Yaskawa INFORM job: test_long_tjr7.JBI

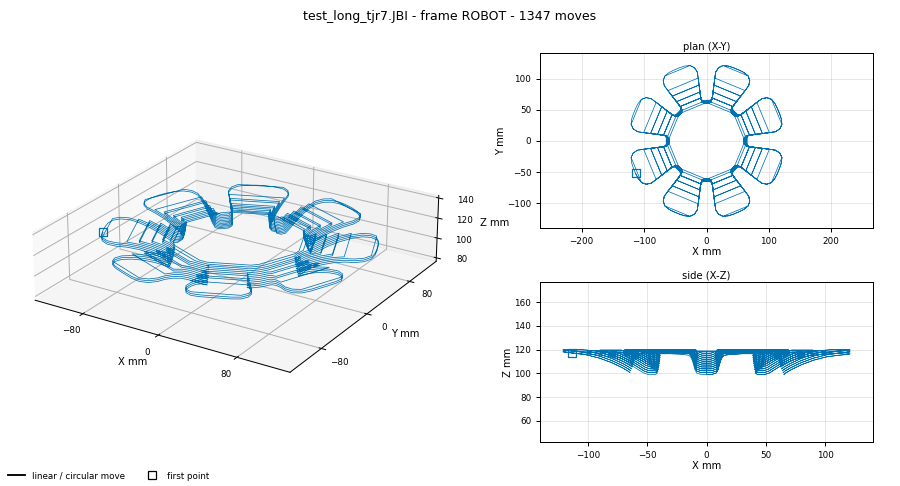
[picture p0: tool path of test_long_tjr7.JBI in frame ROBOT, 1347 of 1348 moves have a stored position in this frame; points joined in program order, loops and branches not executed]
version: 0
/JOB
//NAME test_long
//POS
///NPOS 48,0,0,2,0,0
///TOOL 1
///POSTYPE ROBOT
///RECTAN
///RCONF 1,0,0,0,0,0,0,0,0,0,0,0,0,0,0,0,0,0,0,0,0,0,0,0
C00000=-117.180,-43.520,117.250,-0.0000,-0.0000,1.0000
C00001=-113.630,-52.090,117.250,-0.0000,-0.0000,1.0000
C00002=-109.550,-60.200,116.900,-0.0000,-0.0000,1.0000
C00003=-104.240,-66.670,116.350,-0.0000,-0.0100,1.0000
C00004=-96.760,-69.360,115.810,-0.0000,-0.0200,1.0000
C00005=-88.650,-67.660,115.130,0.0100,-0.0300,1.0000
C00006=-80.860,-61.910,113.810,0.0200,-0.0300,1.0000
C00007=-72.270,-55.220,111.040,0.0200,-0.0300,1.0000
C00008=-64.140,-48.820,107.190,0.0300,-0.0400,1.0000
C00009=-57.630,-43.750,103.240,0.0200,-0.0300,1.0000
C00010=-52.970,-41.300,100.260,-0.0100,0.2100,0.9800
C00011=-49.290,-42.870,99.050,0.2400,0.3300,0.9100
C00012=-47.340,-44.830,99.000,0.3100,0.2900,0.9100
C00013=-46.090,-46.090,99.040,0.3000,0.3000,0.9100
C00014=-44.830,-47.340,99.000,0.2900,0.3100,0.9100
C00015=-42.870,-49.290,99.050,0.3300,0.2400,0.9100
C00016=-41.300,-52.970,100.260,0.2100,-0.0100,0.9800
C00017=-43.750,-57.630,103.240,-0.0300,0.0200,1.0000
C00018=-48.820,-64.140,107.190,-0.0400,0.0300,1.0000
C00019=-55.220,-72.270,111.040,-0.0300,0.0200,1.0000
C00020=-61.910,-80.860,113.810,-0.0300,0.0200,1.0000
C00021=-67.660,-88.650,115.130,-0.0300,0.0100,1.0000
C00022=-69.360,-96.760,115.810,-0.0200,-0.0000,1.0000
C00023=-66.670,-104.240,116.350,-0.0100,-0.0000,1.0000
C00024=-60.200,-109.550,116.900,-0.0000,-0.0000,1.0000
C00025=-52.090,-113.630,117.250,-0.0000,-0.0000,1.0000
C00026=-43.520,-117.180,117.250,-0.0000,-0.0000,1.0000
C00027=-34.900,-120.030,116.900,-0.0000,-0.0000,1.0000
C00028=-26.560,-120.850,116.350,0.0000,-0.0100,1.0000
C00029=-19.380,-117.470,115.810,0.0100,-0.0100,1.0000
C00030=-14.840,-110.530,115.130,0.0300,-0.0100,1.0000
C00031=-13.400,-100.950,113.810,0.0300,-0.0000,1.0000
C00032=-12.060,-90.150,111.040,0.0400,-0.0100,1.0000
C00033=-10.830,-79.870,107.190,0.0400,-0.0100,1.0000
C00034=-9.820,-71.690,103.240,0.0400,-0.0100,1.0000
C00035=-8.250,-66.660,100.260,-0.1600,0.1400,0.9800
C00036=-4.540,-65.170,99.050,-0.0600,0.4000,0.9100
C00037=-1.770,-65.170,99.000,0.0100,0.4200,0.9100
C00038=0.000,-65.190,99.040,-0.0000,0.4200,0.9100
C00039=0.000,-65.190,99.040,-0.0000,0.4200,0.9100
C00040=1.770,-65.170,99.000,-0.0100,0.4200,0.9100
C00041=4.540,-65.170,99.050,0.0600,0.4000,0.9100
C00042=8.250,-66.660,100.260,0.1600,0.1400,0.9800
C00043=9.820,-71.690,103.240,-0.0400,-0.0100,1.0000
C00044=10.830,-79.870,107.190,-0.0400,-0.0100,1.0000
C00045=12.060,-90.150,111.040,-0.0400,-0.0100,1.0000
C00046=13.400,-100.950,113.810,-0.0300,-0.0000,1.0000
C00047=14.840,-110.530,115.130,-0.0300,-0.0100,1.0000
C00048=19.380,-117.470,115.810,-0.0100,-0.0100,1.0000
C00049=26.560,-120.850,116.350,-0.0000,-0.0100,1.0000
C00050=34.900,-120.030,116.900,0.0000,-0.0000,1.0000
C00051=43.520,-117.180,117.250,0.0000,-0.0000,1.0000
C00052=52.090,-113.630,117.250,0.0000,-0.0000,1.0000
C00053=60.200,-109.550,116.900,0.0000,-0.0000,1.0000
C00054=66.670,-104.240,116.350,0.0100,-0.0000,1.0000
C00055=69.360,-96.760,115.810,0.0200,-0.0000,1.0000
C00056=67.660,-88.650,115.130,0.0300,0.0100,1.0000
C00057=61.910,-80.860,113.810,0.0300,0.0200,1.0000
C00058=55.220,-72.270,111.040,0.0300,0.0200,1.0000
C00059=48.820,-64.140,107.190,0.0400,0.0300,1.0000
C00060=43.750,-57.630,103.240,0.0300,0.0200,1.0000
C00061=41.300,-52.970,100.260,-0.2100,-0.0100,0.9800
C00062=42.870,-49.290,99.050,-0.3300,0.2400,0.9100
C00063=44.830,-47.340,99.000,-0.2900,0.3100,0.9100
C00064=46.090,-46.090,99.040,-0.3000,0.3000,0.9100
C00065=47.340,-44.830,99.000,-0.3100,0.2900,0.9100
C00066=49.290,-42.870,99.050,-0.2400,0.3300,0.9100
C00067=52.970,-41.300,100.260,0.0100,0.2100,0.9800
C00068=57.630,-43.750,103.240,-0.0200,-0.0300,1.0000
C00069=64.140,-48.820,107.190,-0.0300,-0.0400,1.0000
C00070=72.270,-55.220,111.040,-0.0200,-0.0300,1.0000
C00071=80.860,-61.910,113.810,-0.0200,-0.0300,1.0000
C00072=88.650,-67.660,115.130,-0.0100,-0.0300,1.0000
C00073=96.760,-69.360,115.810,0.0000,-0.0200,1.0000
C00074=104.240,-66.670,116.350,0.0000,-0.0100,1.0000
C00075=109.550,-60.200,116.900,0.0000,-0.0000,1.0000
C00076=113.630,-52.090,117.250,0.0000,-0.0000,1.0000
C00077=117.180,-43.520,117.250,0.0000,-0.0000,1.0000
C00078=120.030,-34.900,116.900,0.0000,-0.0000,1.0000
C00079=120.850,-26.560,116.350,0.0100,0.0000,1.0000
C00080=117.470,-19.380,115.810,0.0100,0.0100,1.0000
C00081=110.530,-14.840,115.130,0.0100,0.0300,1.0000
C00082=100.950,-13.400,113.810,0.0000,0.0300,1.0000
C00083=90.150,-12.060,111.040,0.0100,0.0400,1.0000
C00084=79.870,-10.830,107.190,0.0100,0.0400,1.0000
C00085=71.690,-9.820,103.240,0.0100,0.0400,1.0000
C00086=66.660,-8.250,100.260,-0.1400,-0.1600,0.9800
C00087=65.170,-4.540,99.050,-0.4000,-0.0600,0.9100
C00088=65.170,-1.770,99.000,-0.4200,0.0100,0.9100
C00089=65.190,0.000,99.040,-0.4200,-0.0000,0.9100
C00090=65.170,1.770,99.000,-0.4200,-0.0100,0.9100
C00091=65.170,4.540,99.050,-0.4000,0.0600,0.9100
C00092=66.660,8.250,100.260,-0.1400,0.1600,0.9800
C00093=71.690,9.820,103.240,0.0100,-0.0400,1.0000
C00094=79.870,10.830,107.190,0.0100,-0.0400,1.0000
C00095=90.150,12.060,111.040,0.0100,-0.0400,1.0000
C00096=100.950,13.400,113.810,0.0000,-0.0300,1.0000
C00097=110.530,14.840,115.130,0.0100,-0.0300,1.0000
C00098=117.470,19.380,115.810,0.0100,-0.0100,1.0000
C00099=120.850,26.560,116.350,0.0100,-0.0000,1.0000
C00100=120.030,34.900,116.900,0.0000,0.0000,1.0000
C00101=117.180,43.520,117.250,0.0000,0.0000,1.0000
C00102=113.630,52.090,117.250,0.0000,0.0000,1.0000
C00103=109.550,60.200,116.900,0.0000,0.0000,1.0000
C00104=104.240,66.670,116.350,0.0000,0.0100,1.0000
C00105=96.760,69.360,115.810,0.0000,0.0200,1.0000
C00106=88.650,67.660,115.130,-0.0100,0.0300,1.0000
C00107=80.860,61.910,113.810,-0.0200,0.0300,1.0000
C00108=72.270,55.220,111.040,-0.0200,0.0300,1.0000
C00109=64.140,48.820,107.190,-0.0300,0.0400,1.0000
C00110=57.630,43.750,103.240,-0.0200,0.0300,1.0000
C00111=52.970,41.300,100.260,0.0100,-0.2100,0.9800
C00112=49.290,42.870,99.050,-0.2400,-0.3300,0.9100
C00113=47.340,44.830,99.000,-0.3100,-0.2900,0.9100
C00114=46.090,46.090,99.040,-0.3000,-0.3000,0.9100
C00115=44.830,47.340,99.000,-0.2900,-0.3100,0.9100
C00116=42.870,49.290,99.050,-0.3300,-0.2400,0.9100
C00117=41.300,52.970,100.260,-0.2100,0.0100,0.9800
C00118=43.750,57.630,103.240,0.0300,-0.0200,1.0000
C00119=48.820,64.140,107.190,0.0400,-0.0300,1.0000
C00120=55.220,72.270,111.040,0.0300,-0.0200,1.0000
C00121=61.910,80.860,113.810,0.0300,-0.0200,1.0000
C00122=67.660,88.650,115.130,0.0300,-0.0100,1.0000
C00123=69.360,96.760,115.810,0.0200,0.0000,1.0000
C00124=66.670,104.240,116.350,0.0100,0.0000,1.0000
C00125=60.200,109.550,116.900,0.0000,0.0000,1.0000
C00126=52.090,113.630,117.250,0.0000,0.0000,1.0000
C00127=43.520,117.180,117.250,0.0000,0.0000,1.0000
C00128=34.900,120.030,116.900,0.0000,0.0000,1.0000
C00129=26.560,120.850,116.350,-0.0000,0.0100,1.0000
C00130=19.380,117.470,115.810,-0.0100,0.0100,1.0000
C00131=14.840,110.530,115.130,-0.0300,0.0100,1.0000
C00132=13.400,100.950,113.810,-0.0300,0.0000,1.0000
C00133=12.060,90.150,111.040,-0.0400,0.0100,1.0000
C00134=10.830,79.870,107.190,-0.0400,0.0100,1.0000
C00135=9.820,71.690,103.240,-0.0400,0.0100,1.0000
C00136=8.250,66.660,100.260,0.1600,-0.1400,0.9800
C00137=4.540,65.170,99.050,0.0600,-0.4000,0.9100
C00138=1.770,65.170,99.000,-0.0100,-0.4200,0.9100
C00139=0.000,65.190,99.040,-0.0000,-0.4200,0.9100
C00140=0.000,64.490,100.590,-0.0000,-0.4000,0.9200
C00141=1.710,64.480,100.550,-0.0100,-0.4000,0.9200
C00142=4.440,64.480,100.600,0.0600,-0.3800,0.9200
C00143=8.120,66.020,101.830,0.1500,-0.1200,0.9800
C00144=9.680,71.190,104.850,-0.0300,0.0000,1.0000
C00145=10.710,79.550,108.860,-0.0400,0.0100,1.0000
C00146=11.970,89.980,112.730,-0.0300,0.0000,1.0000
C00147=13.340,100.880,115.510,-0.0300,0.0000,1.0000
C00148=14.790,110.500,116.830,-0.0200,0.0100,1.0000
C00149=19.340,117.460,117.510,-0.0100,0.0100,1.0000
C00150=26.540,120.860,118.050,-0.0000,0.0000,1.0000
C00151=34.880,120.030,118.600,0.0000,0.0000,1.0000
C00152=43.510,117.180,118.950,0.0000,0.0000,1.0000
C00153=52.090,113.630,118.950,0.0000,0.0000,1.0000
C00154=60.210,109.540,118.600,0.0000,0.0000,1.0000
C00155=66.700,104.220,118.050,0.0000,0.0000,1.0000
C00156=69.380,96.730,117.510,0.0100,0.0000,1.0000
C00157=67.680,88.590,116.830,0.0200,-0.0100,1.0000
C00158=61.900,80.770,115.510,0.0200,-0.0200,1.0000
C00159=55.160,72.090,112.730,0.0300,-0.0200,1.0000
C00160=48.670,63.820,108.860,0.0300,-0.0200,1.0000
C00161=43.490,57.190,104.850,0.0300,-0.0200,1.0000
C00162=40.940,52.430,101.830,-0.1900,0.0200,0.9800
C00163=42.460,48.730,100.600,-0.3100,-0.2300,0.9200
C00164=44.380,46.800,100.550,-0.2700,-0.2900,0.9200
C00165=45.600,45.600,100.590,-0.2800,-0.2800,0.9200
C00166=46.800,44.380,100.550,-0.2900,-0.2700,0.9200
C00167=48.730,42.460,100.600,-0.2300,-0.3100,0.9200
C00168=52.430,40.940,101.830,0.0200,-0.1900,0.9800
C00169=57.190,43.490,104.850,-0.0200,0.0300,1.0000
C00170=63.820,48.670,108.860,-0.0200,0.0300,1.0000
C00171=72.090,55.160,112.730,-0.0200,0.0300,1.0000
C00172=80.770,61.900,115.510,-0.0200,0.0200,1.0000
C00173=88.590,67.680,116.830,-0.0100,0.0200,1.0000
C00174=96.730,69.380,117.510,0.0000,0.0100,1.0000
C00175=104.220,66.700,118.050,0.0000,0.0000,1.0000
C00176=109.540,60.210,118.600,0.0000,0.0000,1.0000
C00177=113.630,52.090,118.950,0.0000,0.0000,1.0000
C00178=117.180,43.510,118.950,0.0000,0.0000,1.0000
C00179=120.030,34.880,118.600,0.0000,0.0000,1.0000
C00180=120.860,26.540,118.050,0.0000,-0.0000,1.0000
C00181=117.460,19.340,117.510,0.0100,-0.0100,1.0000
C00182=110.500,14.790,116.830,0.0100,-0.0200,1.0000
C00183=100.880,13.340,115.510,0.0000,-0.0300,1.0000
C00184=89.980,11.970,112.730,0.0000,-0.0300,1.0000
C00185=79.550,10.710,108.860,0.0100,-0.0400,1.0000
C00186=71.190,9.680,104.850,0.0000,-0.0300,1.0000
C00187=66.020,8.120,101.830,-0.1200,0.1500,0.9800
C00188=64.480,4.440,100.600,-0.3800,0.0600,0.9200
C00189=64.480,1.710,100.550,-0.4000,-0.0100,0.9200
C00190=64.490,0.000,100.590,-0.4000,-0.0000,0.9200
C00191=64.480,-1.710,100.550,-0.4000,0.0100,0.9200
C00192=64.480,-4.440,100.600,-0.3800,-0.0600,0.9200
C00193=66.020,-8.120,101.830,-0.1200,-0.1500,0.9800
C00194=71.190,-9.680,104.850,0.0000,0.0300,1.0000
C00195=79.550,-10.710,108.860,0.0100,0.0400,1.0000
C00196=89.980,-11.970,112.730,0.0000,0.0300,1.0000
C00197=100.880,-13.340,115.510,0.0000,0.0300,1.0000
C00198=110.500,-14.790,116.830,0.0100,0.0200,1.0000
C00199=117.460,-19.340,117.510,0.0100,0.0100,1.0000
C00200=120.860,-26.540,118.050,0.0000,0.0000,1.0000
C00201=120.030,-34.880,118.600,0.0000,-0.0000,1.0000
C00202=117.180,-43.510,118.950,0.0000,-0.0000,1.0000
C00203=113.630,-52.090,118.950,0.0000,-0.0000,1.0000
C00204=109.540,-60.210,118.600,0.0000,-0.0000,1.0000
C00205=104.220,-66.700,118.050,0.0000,-0.0000,1.0000
C00206=96.730,-69.380,117.510,0.0000,-0.0100,1.0000
C00207=88.590,-67.680,116.830,-0.0100,-0.0200,1.0000
C00208=80.770,-61.900,115.510,-0.0200,-0.0200,1.0000
C00209=72.090,-55.160,112.730,-0.0200,-0.0300,1.0000
C00210=63.820,-48.670,108.860,-0.0200,-0.0300,1.0000
C00211=57.190,-43.490,104.850,-0.0200,-0.0300,1.0000
C00212=52.430,-40.940,101.830,0.0200,0.1900,0.9800
C00213=48.730,-42.460,100.600,-0.2300,0.3100,0.9200
C00214=46.800,-44.380,100.550,-0.2900,0.2700,0.9200
C00215=45.600,-45.600,100.590,-0.2800,0.2800,0.9200
C00216=44.380,-46.800,100.550,-0.2700,0.2900,0.9200
C00217=42.460,-48.730,100.600,-0.3100,0.2300,0.9200
C00218=40.940,-52.430,101.830,-0.1900,-0.0200,0.9800
C00219=43.490,-57.190,104.850,0.0300,0.0200,1.0000
C00220=48.670,-63.820,108.860,0.0300,0.0200,1.0000
C00221=55.160,-72.090,112.730,0.0300,0.0200,1.0000
C00222=61.900,-80.770,115.510,0.0200,0.0200,1.0000
C00223=67.680,-88.590,116.830,0.0200,0.0100,1.0000
C00224=69.380,-96.730,117.510,0.0100,-0.0000,1.0000
C00225=66.700,-104.220,118.050,0.0000,-0.0000,1.0000
C00226=60.210,-109.540,118.600,0.0000,-0.0000,1.0000
C00227=52.090,-113.630,118.950,0.0000,-0.0000,1.0000
C00228=43.510,-117.180,118.950,0.0000,-0.0000,1.0000
C00229=34.880,-120.030,118.600,0.0000,-0.0000,1.0000
C00230=26.540,-120.860,118.050,-0.0000,-0.0000,1.0000
C00231=19.340,-117.460,117.510,-0.0100,-0.0100,1.0000
C00232=14.790,-110.500,116.830,-0.0200,-0.0100,1.0000
C00233=13.340,-100.880,115.510,-0.0300,-0.0000,1.0000
C00234=11.970,-89.980,112.730,-0.0300,-0.0000,1.0000
C00235=10.710,-79.550,108.860,-0.0400,-0.0100,1.0000
C00236=9.680,-71.190,104.850,-0.0300,-0.0000,1.0000
C00237=8.120,-66.020,101.830,0.1500,0.1200,0.9800
C00238=4.440,-64.480,100.600,0.0600,0.3800,0.9200
C00239=1.710,-64.480,100.550,-0.0100,0.4000,0.9200
C00240=0.000,-64.490,100.590,-0.0000,0.4000,0.9200
C00241=0.000,-64.490,100.590,-0.0000,0.4000,0.9200
C00242=-1.710,-64.480,100.550,0.0100,0.4000,0.9200
C00243=-4.440,-64.480,100.600,-0.0600,0.3800,0.9200
C00244=-8.120,-66.020,101.830,-0.1500,0.1200,0.9800
C00245=-9.680,-71.190,104.850,0.0300,-0.0000,1.0000
C00246=-10.710,-79.550,108.860,0.0400,-0.0100,1.0000
C00247=-11.970,-89.980,112.730,0.0300,-0.0000,1.0000
C00248=-13.340,-100.880,115.510,0.0300,-0.0000,1.0000
C00249=-14.790,-110.500,116.830,0.0200,-0.0100,1.0000
C00250=-19.340,-117.460,117.510,0.0100,-0.0100,1.0000
C00251=-26.540,-120.860,118.050,0.0000,-0.0000,1.0000
C00252=-34.880,-120.030,118.600,-0.0000,-0.0000,1.0000
C00253=-43.510,-117.180,118.950,-0.0000,-0.0000,1.0000
C00254=-52.090,-113.630,118.950,-0.0000,-0.0000,1.0000
C00255=-60.210,-109.540,118.600,-0.0000,-0.0000,1.0000
C00256=-66.700,-104.220,118.050,-0.0000,-0.0000,1.0000
C00257=-69.380,-96.730,117.510,-0.0100,-0.0000,1.0000
C00258=-67.680,-88.590,116.830,-0.0200,0.0100,1.0000
C00259=-61.900,-80.770,115.510,-0.0200,0.0200,1.0000
C00260=-55.160,-72.090,112.730,-0.0300,0.0200,1.0000
C00261=-48.670,-63.820,108.860,-0.0300,0.0200,1.0000
C00262=-43.490,-57.190,104.850,-0.0300,0.0200,1.0000
C00263=-40.940,-52.430,101.830,0.1900,-0.0200,0.9800
C00264=-42.460,-48.730,100.600,0.3100,0.2300,0.9200
C00265=-44.380,-46.800,100.550,0.2700,0.2900,0.9200
C00266=-45.600,-45.600,100.590,0.2800,0.2800,0.9200
C00267=-46.800,-44.380,100.550,0.2900,0.2700,0.9200
C00268=-48.730,-42.460,100.600,0.2300,0.3100,0.9200
C00269=-52.430,-40.940,101.830,-0.0200,0.1900,0.9800
C00270=-57.190,-43.490,104.850,0.0200,-0.0300,1.0000
C00271=-63.820,-48.670,108.860,0.0200,-0.0300,1.0000
C00272=-72.090,-55.160,112.730,0.0200,-0.0300,1.0000
C00273=-80.770,-61.900,115.510,0.0200,-0.0200,1.0000
C00274=-88.590,-67.680,116.830,0.0100,-0.0200,1.0000
C00275=-96.730,-69.380,117.510,-0.0000,-0.0100,1.0000
C00276=-104.220,-66.700,118.050,-0.0000,-0.0000,1.0000
C00277=-109.540,-60.210,118.600,-0.0000,-0.0000,1.0000
C00278=-113.630,-52.090,118.950,-0.0000,-0.0000,1.0000
C00279=-117.180,-43.510,118.950,-0.0000,-0.0000,1.0000
C00280=-120.030,-34.880,118.600,-0.0000,-0.0000,1.0000
C00281=-120.860,-26.540,118.050,-0.0000,0.0000,1.0000
C00282=-117.460,-19.340,117.510,-0.0100,0.0100,1.0000
C00283=-110.500,-14.790,116.830,-0.0100,0.0200,1.0000
C00284=-100.880,-13.340,115.510,-0.0000,0.0300,1.0000
C00285=-89.980,-11.970,112.730,-0.0000,0.0300,1.0000
C00286=-79.550,-10.710,108.860,-0.0100,0.0400,1.0000
C00287=-71.190,-9.680,104.850,-0.0000,0.0300,1.0000
C00288=-66.020,-8.120,101.830,0.1200,-0.1500,0.9800
C00289=-64.480,-4.440,100.600,0.3800,-0.0600,0.9200
C00290=-64.480,-1.710,100.550,0.4000,0.0100,0.9200
C00291=-64.490,0.000,100.590,0.4000,0.0000,0.9200
C00292=-64.480,1.710,100.550,0.4000,-0.0100,0.9200
C00293=-64.480,4.440,100.600,0.3800,0.0600,0.9200
C00294=-66.020,8.120,101.830,0.1200,0.1500,0.9800
C00295=-71.190,9.680,104.850,-0.0000,-0.0300,1.0000
C00296=-79.550,10.710,108.860,-0.0100,-0.0400,1.0000
C00297=-89.980,11.970,112.730,-0.0000,-0.0300,1.0000
C00298=-100.880,13.340,115.510,-0.0000,-0.0300,1.0000
C00299=-110.500,14.790,116.830,-0.0100,-0.0200,1.0000
C00300=-117.460,19.340,117.510,-0.0100,-0.0100,1.0000
C00301=-120.860,26.540,118.050,-0.0000,-0.0000,1.0000
C00302=-120.030,34.880,118.600,-0.0000,0.0000,1.0000
C00303=-117.180,43.510,118.950,-0.0000,0.0000,1.0000
C00304=-113.630,52.090,118.950,-0.0000,0.0000,1.0000
C00305=-109.540,60.210,118.600,-0.0000,0.0000,1.0000
C00306=-104.220,66.700,118.050,-0.0000,0.0000,1.0000
C00307=-96.730,69.380,117.510,-0.0000,0.0100,1.0000
C00308=-88.590,67.680,116.830,0.0100,0.0200,1.0000
C00309=-80.770,61.900,115.510,0.0200,0.0200,1.0000
C00310=-72.090,55.160,112.730,0.0200,0.0300,1.0000
C00311=-63.820,48.670,108.860,0.0200,0.0300,1.0000
C00312=-57.190,43.490,104.850,0.0200,0.0300,1.0000
C00313=-52.430,40.940,101.830,-0.0200,-0.1900,0.9800
C00314=-48.730,42.460,100.600,0.2300,-0.3100,0.9200
C00315=-46.800,44.380,100.550,0.2900,-0.2700,0.9200
C00316=-45.600,45.600,100.590,0.2800,-0.2800,0.9200
C00317=-44.380,46.800,100.550,0.2700,-0.2900,0.9200
C00318=-42.460,48.730,100.600,0.3100,-0.2300,0.9200
C00319=-40.940,52.430,101.830,0.1900,0.0200,0.9800
C00320=-43.490,57.190,104.850,-0.0300,-0.0200,1.0000
C00321=-48.670,63.820,108.860,-0.0300,-0.0200,1.0000
C00322=-55.160,72.090,112.730,-0.0300,-0.0200,1.0000
C00323=-61.900,80.770,115.510,-0.0200,-0.0200,1.0000
C00324=-67.680,88.590,116.830,-0.0200,-0.0100,1.0000
C00325=-69.380,96.730,117.510,-0.0100,0.0000,1.0000
C00326=-66.700,104.220,118.050,-0.0000,0.0000,1.0000
C00327=-60.210,109.540,118.600,-0.0000,0.0000,1.0000
C00328=-52.090,113.630,118.950,-0.0000,0.0000,1.0000
C00329=-43.510,117.180,118.950,-0.0000,0.0000,1.0000
C00330=-34.880,120.030,118.600,-0.0000,0.0000,1.0000
C00331=-26.540,120.860,118.050,0.0000,0.0000,1.0000
C00332=-19.340,117.460,117.510,0.0100,0.0100,1.0000
C00333=-14.790,110.500,116.830,0.0200,0.0100,1.0000
C00334=-13.340,100.880,115.510,0.0300,0.0000,1.0000
C00335=-11.970,89.980,112.730,0.0300,0.0000,1.0000
C00336=-10.710,79.550,108.860,0.0400,0.0100,1.0000
C00337=-9.680,71.190,104.850,0.0300,0.0000,1.0000
C00338=-8.120,66.020,101.830,-0.1500,-0.1200,0.9800
C00339=-4.440,64.480,100.600,-0.0600,-0.3800,0.9200
C00340=-1.710,64.480,100.550,0.0100,-0.4000,0.9200
C00341=0.000,64.490,100.590,-0.0000,-0.4000,0.9200
C00342=0.000,63.830,102.150,-0.0000,-0.3800,0.9300
C00343=-1.650,63.820,102.110,0.0100,-0.3800,0.9300
C00344=-4.330,63.820,102.170,-0.0600,-0.3600,0.9300
C00345=-8.010,65.430,103.420,-0.1300,-0.1100,0.9800
C00346=-9.560,70.730,106.490,0.0300,0.0000,1.0000
C00347=-10.610,79.260,110.530,0.0300,0.0000,1.0000
C00348=-11.900,89.840,114.420,0.0300,0.0000,1.0000
C00349=-13.300,100.830,117.210,0.0200,0.0000,1.0000
C00350=-14.760,110.480,118.530,0.0100,0.0000,1.0000
C00351=-19.320,117.460,119.210,0.0000,0.0000,1.0000
C00352=-26.530,120.860,119.750,0.0000,0.0000,1.0000
C00353=-66.700,104.220,119.750,-0.0000,0.0000,1.0000
C00354=-69.390,96.720,119.210,-0.0000,0.0000,1.0000
C00355=-67.690,88.560,118.530,-0.0100,-0.0000,1.0000
C00356=-61.890,80.700,117.210,-0.0100,-0.0100,1.0000
C00357=-55.110,71.950,114.420,-0.0200,-0.0200,1.0000
C00358=-48.550,63.550,110.530,-0.0300,-0.0200,1.0000
C00359=-43.250,56.780,106.490,-0.0300,-0.0200,1.0000
C00360=-40.600,51.930,103.420,0.1700,0.0200,0.9800
C00361=-42.070,48.200,102.170,0.2900,-0.2100,0.9300
C00362=-43.960,46.290,102.110,0.2600,-0.2700,0.9300
C00363=-45.130,45.130,102.150,0.2700,-0.2700,0.9300
C00364=-46.290,43.960,102.110,0.2700,-0.2600,0.9300
C00365=-48.200,42.070,102.170,0.2100,-0.2900,0.9300
C00366=-51.930,40.600,103.420,-0.0200,-0.1700,0.9800
C00367=-56.780,43.250,106.490,0.0200,0.0300,1.0000
C00368=-63.550,48.550,110.530,0.0200,0.0300,1.0000
C00369=-71.950,55.110,114.420,0.0200,0.0200,1.0000
C00370=-80.700,61.890,117.210,0.0100,0.0100,1.0000
C00371=-88.560,67.690,118.530,0.0000,0.0100,1.0000
C00372=-96.720,69.390,119.210,-0.0000,0.0000,1.0000
C00373=-104.220,66.700,119.750,-0.0000,0.0000,1.0000
C00374=-120.860,26.530,119.750,-0.0000,-0.0000,1.0000
C00375=-117.460,19.320,119.210,-0.0000,-0.0000,1.0000
C00376=-110.480,14.760,118.530,-0.0000,-0.0100,1.0000
C00377=-100.830,13.300,117.210,-0.0000,-0.0200,1.0000
C00378=-89.840,11.900,114.420,-0.0000,-0.0300,1.0000
C00379=-79.260,10.610,110.530,-0.0000,-0.0300,1.0000
C00380=-70.730,9.560,106.490,-0.0000,-0.0300,1.0000
C00381=-65.430,8.010,103.420,0.1100,0.1300,0.9800
C00382=-63.820,4.330,102.170,0.3600,0.0600,0.9300
C00383=-63.820,1.650,102.110,0.3800,-0.0100,0.9300
C00384=-63.830,0.000,102.150,0.3800,0.0000,0.9300
C00385=-63.820,-1.650,102.110,0.3800,0.0100,0.9300
C00386=-63.820,-4.330,102.170,0.3600,-0.0600,0.9300
C00387=-65.430,-8.010,103.420,0.1100,-0.1300,0.9800
C00388=-70.730,-9.560,106.490,-0.0000,0.0300,1.0000
C00389=-79.260,-10.610,110.530,-0.0000,0.0300,1.0000
C00390=-89.840,-11.900,114.420,-0.0000,0.0300,1.0000
C00391=-100.830,-13.300,117.210,-0.0000,0.0200,1.0000
C00392=-110.480,-14.760,118.530,-0.0000,0.0100,1.0000
C00393=-117.460,-19.320,119.210,-0.0000,0.0000,1.0000
C00394=-120.860,-26.530,119.750,-0.0000,0.0000,1.0000
C00395=-104.220,-66.700,119.750,-0.0000,-0.0000,1.0000
C00396=-96.720,-69.390,119.210,-0.0000,-0.0000,1.0000
C00397=-88.560,-67.690,118.530,0.0000,-0.0100,1.0000
C00398=-80.700,-61.890,117.210,0.0100,-0.0100,1.0000
C00399=-71.950,-55.110,114.420,0.0200,-0.0200,1.0000
C00400=-63.550,-48.550,110.530,0.0200,-0.0300,1.0000
C00401=-56.780,-43.250,106.490,0.0200,-0.0300,1.0000
C00402=-51.930,-40.600,103.420,-0.0200,0.1700,0.9800
C00403=-48.200,-42.070,102.170,0.2100,0.2900,0.9300
C00404=-46.290,-43.960,102.110,0.2700,0.2600,0.9300
C00405=-45.130,-45.130,102.150,0.2700,0.2700,0.9300
C00406=-43.960,-46.290,102.110,0.2600,0.2700,0.9300
C00407=-42.070,-48.200,102.170,0.2900,0.2100,0.9300
C00408=-40.600,-51.930,103.420,0.1700,-0.0200,0.9800
C00409=-43.250,-56.780,106.490,-0.0300,0.0200,1.0000
C00410=-48.550,-63.550,110.530,-0.0300,0.0200,1.0000
C00411=-55.110,-71.950,114.420,-0.0200,0.0200,1.0000
C00412=-61.890,-80.700,117.210,-0.0100,0.0100,1.0000
C00413=-67.690,-88.560,118.530,-0.0100,0.0000,1.0000
C00414=-69.390,-96.720,119.210,-0.0000,-0.0000,1.0000
C00415=-66.700,-104.220,119.750,-0.0000,-0.0000,1.0000
C00416=-26.530,-120.860,119.750,0.0000,-0.0000,1.0000
C00417=-19.320,-117.460,119.210,0.0000,-0.0000,1.0000
C00418=-14.760,-110.480,118.530,0.0100,-0.0000,1.0000
C00419=-13.300,-100.830,117.210,0.0200,-0.0000,1.0000
C00420=-11.900,-89.840,114.420,0.0300,-0.0000,1.0000
C00421=-10.610,-79.260,110.530,0.0300,-0.0000,1.0000
C00422=-9.560,-70.730,106.490,0.0300,-0.0000,1.0000
C00423=-8.010,-65.430,103.420,-0.1300,0.1100,0.9800
C00424=-4.330,-63.820,102.170,-0.0600,0.3600,0.9300
C00425=-1.650,-63.820,102.110,0.0100,0.3800,0.9300
C00426=0.000,-63.830,102.150,-0.0000,0.3800,0.9300
C00427=0.000,-63.830,102.150,-0.0000,0.3800,0.9300
C00428=1.650,-63.820,102.110,-0.0100,0.3800,0.9300
C00429=4.330,-63.820,102.170,0.0600,0.3600,0.9300
C00430=8.010,-65.430,103.420,0.1300,0.1100,0.9800
C00431=9.560,-70.730,106.490,-0.0300,-0.0000,1.0000
C00432=10.610,-79.260,110.530,-0.0300,-0.0000,1.0000
C00433=11.900,-89.840,114.420,-0.0300,-0.0000,1.0000
C00434=13.300,-100.830,117.210,-0.0200,-0.0000,1.0000
C00435=14.760,-110.480,118.530,-0.0100,-0.0000,1.0000
C00436=19.320,-117.460,119.210,-0.0000,-0.0000,1.0000
C00437=26.530,-120.860,119.750,-0.0000,-0.0000,1.0000
C00438=66.700,-104.220,119.750,0.0000,-0.0000,1.0000
C00439=69.390,-96.720,119.210,0.0000,-0.0000,1.0000
C00440=67.690,-88.560,118.530,0.0100,0.0000,1.0000
C00441=61.890,-80.700,117.210,0.0100,0.0100,1.0000
C00442=55.110,-71.950,114.420,0.0200,0.0200,1.0000
C00443=48.550,-63.550,110.530,0.0300,0.0200,1.0000
C00444=43.250,-56.780,106.490,0.0300,0.0200,1.0000
C00445=40.600,-51.930,103.420,-0.1700,-0.0200,0.9800
C00446=42.070,-48.200,102.170,-0.2900,0.2100,0.9300
C00447=43.960,-46.290,102.110,-0.2600,0.2700,0.9300
C00448=45.130,-45.130,102.150,-0.2700,0.2700,0.9300
C00449=46.290,-43.960,102.110,-0.2700,0.2600,0.9300
C00450=48.200,-42.070,102.170,-0.2100,0.2900,0.9300
C00451=51.930,-40.600,103.420,0.0200,0.1700,0.9800
C00452=56.780,-43.250,106.490,-0.0200,-0.0300,1.0000
C00453=63.550,-48.550,110.530,-0.0200,-0.0300,1.0000
C00454=71.950,-55.110,114.420,-0.0200,-0.0200,1.0000
C00455=80.700,-61.890,117.210,-0.0100,-0.0100,1.0000
C00456=88.560,-67.690,118.530,-0.0000,-0.0100,1.0000
C00457=96.720,-69.390,119.210,0.0000,-0.0000,1.0000
C00458=104.220,-66.700,119.750,0.0000,-0.0000,1.0000
C00459=120.860,-26.530,119.750,0.0000,0.0000,1.0000
C00460=117.460,-19.320,119.210,0.0000,0.0000,1.0000
C00461=110.480,-14.760,118.530,0.0000,0.0100,1.0000
C00462=100.830,-13.300,117.210,0.0000,0.0200,1.0000
C00463=89.840,-11.900,114.420,0.0000,0.0300,1.0000
C00464=79.260,-10.610,110.530,0.0000,0.0300,1.0000
C00465=70.730,-9.560,106.490,0.0000,0.0300,1.0000
C00466=65.430,-8.010,103.420,-0.1100,-0.1300,0.9800
C00467=63.820,-4.330,102.170,-0.3600,-0.0600,0.9300
C00468=63.820,-1.650,102.110,-0.3800,0.0100,0.9300
C00469=63.830,0.000,102.150,-0.3800,-0.0000,0.9300
C00470=63.820,1.650,102.110,-0.3800,-0.0100,0.9300
C00471=63.820,4.330,102.170,-0.3600,0.0600,0.9300
C00472=65.430,8.010,103.420,-0.1100,0.1300,0.9800
C00473=70.730,9.560,106.490,0.0000,-0.0300,1.0000
C00474=79.260,10.610,110.530,0.0000,-0.0300,1.0000
C00475=89.840,11.900,114.420,0.0000,-0.0300,1.0000
C00476=100.830,13.300,117.210,0.0000,-0.0200,1.0000
C00477=110.480,14.760,118.530,0.0000,-0.0100,1.0000
C00478=117.460,19.320,119.210,0.0000,-0.0000,1.0000
C00479=120.860,26.530,119.750,0.0000,-0.0000,1.0000
C00480=104.220,66.700,119.750,0.0000,0.0000,1.0000
C00481=96.720,69.390,119.210,0.0000,0.0000,1.0000
C00482=88.560,67.690,118.530,-0.0000,0.0100,1.0000
C00483=80.700,61.890,117.210,-0.0100,0.0100,1.0000
C00484=71.950,55.110,114.420,-0.0200,0.0200,1.0000
C00485=63.550,48.550,110.530,-0.0200,0.0300,1.0000
C00486=56.780,43.250,106.490,-0.0200,0.0300,1.0000
C00487=51.930,40.600,103.420,0.0200,-0.1700,0.9800
C00488=48.200,42.070,102.170,-0.2100,-0.2900,0.9300
C00489=46.290,43.960,102.110,-0.2700,-0.2600,0.9300
C00490=45.130,45.130,102.150,-0.2700,-0.2700,0.9300
C00491=43.960,46.290,102.110,-0.2600,-0.2700,0.9300
C00492=42.070,48.200,102.170,-0.2900,-0.2100,0.9300
C00493=40.600,51.930,103.420,-0.1700,0.0200,0.9800
C00494=43.250,56.780,106.490,0.0300,-0.0200,1.0000
C00495=48.550,63.550,110.530,0.0300,-0.0200,1.0000
C00496=55.110,71.950,114.420,0.0200,-0.0200,1.0000
C00497=61.890,80.700,117.210,0.0100,-0.0100,1.0000
C00498=67.690,88.560,118.530,0.0100,-0.0000,1.0000
C00499=69.390,96.720,119.210,0.0000,0.0000,1.0000
C00500=66.700,104.220,119.750,0.0000,0.0000,1.0000
C00501=26.530,120.860,119.750,-0.0000,0.0000,1.0000
C00502=19.320,117.460,119.210,-0.0000,0.0000,1.0000
C00503=14.760,110.480,118.530,-0.0100,0.0000,1.0000
C00504=13.300,100.830,117.210,-0.0200,0.0000,1.0000
C00505=11.900,89.840,114.420,-0.0300,0.0000,1.0000
C00506=10.610,79.260,110.530,-0.0300,0.0000,1.0000
C00507=9.560,70.730,106.490,-0.0300,0.0000,1.0000
C00508=8.010,65.430,103.420,0.1300,-0.1100,0.9800
C00509=4.330,63.820,102.170,0.0600,-0.3600,0.9300
C00510=1.650,63.820,102.110,-0.0100,-0.3800,0.9300
C00511=0.000,63.830,102.150,-0.0000,-0.3800,0.9300
C00512=0.000,63.210,103.730,-0.0000,-0.3500,0.9400
C00513=1.590,63.200,103.700,-0.0100,-0.3500,0.9400
C00514=4.240,63.210,103.750,0.0500,-0.3300,0.9400
C00515=7.900,64.870,105.020,0.1200,-0.1000,0.9900
C00516=9.450,70.320,108.130,-0.0300,0.0000,1.0000
C00517=10.520,79.020,112.210,-0.0300,0.0000,1.0000
C00518=11.850,89.740,116.120,-0.0200,0.0000,1.0000
C00519=13.270,100.800,118.910,-0.0100,0.0000,1.0000
C00520=61.890,80.660,118.910,0.0100,-0.0000,1.0000
C00521=55.080,71.840,116.120,0.0100,-0.0100,1.0000
C00522=48.440,63.320,112.210,0.0200,-0.0200,1.0000
C00523=43.040,56.410,108.130,0.0200,-0.0200,1.0000
C00524=40.290,51.460,105.020,-0.1600,0.0200,0.9900
C00525=41.700,47.690,103.750,-0.2700,-0.2000,0.9400
C00526=43.560,45.810,103.700,-0.2400,-0.2600,0.9400
C00527=44.690,44.690,103.730,-0.2500,-0.2500,0.9400
C00528=45.810,43.560,103.700,-0.2600,-0.2400,0.9400
C00529=47.700,41.700,103.750,-0.2000,-0.2700,0.9400
C00530=51.460,40.290,105.020,0.0200,-0.1600,0.9900
C00531=56.410,43.040,108.130,-0.0200,0.0200,1.0000
C00532=63.320,48.440,112.210,-0.0200,0.0200,1.0000
C00533=71.840,55.080,116.120,-0.0100,0.0100,1.0000
C00534=80.660,61.890,118.910,-0.0000,0.0100,1.0000
C00535=100.800,13.270,118.910,0.0000,-0.0100,1.0000
C00536=89.740,11.850,116.120,0.0000,-0.0200,1.0000
C00537=79.020,10.520,112.210,0.0000,-0.0300,1.0000
C00538=70.320,9.450,108.130,0.0000,-0.0300,1.0000
C00539=64.870,7.900,105.020,-0.1000,0.1200,0.9900
C00540=63.210,4.240,103.750,-0.3300,0.0500,0.9400
C00541=63.200,1.590,103.700,-0.3500,-0.0100,0.9400
C00542=63.210,0.000,103.730,-0.3500,-0.0000,0.9400
C00543=63.200,-1.590,103.700,-0.3500,0.0100,0.9400
C00544=63.210,-4.240,103.750,-0.3300,-0.0500,0.9400
C00545=64.870,-7.900,105.020,-0.1000,-0.1200,0.9900
C00546=70.320,-9.450,108.130,0.0000,0.0300,1.0000
C00547=79.020,-10.520,112.210,0.0000,0.0300,1.0000
C00548=89.740,-11.850,116.120,0.0000,0.0200,1.0000
C00549=100.800,-13.270,118.910,0.0000,0.0100,1.0000
C00550=80.660,-61.890,118.910,-0.0000,-0.0100,1.0000
C00551=71.840,-55.080,116.120,-0.0100,-0.0100,1.0000
C00552=63.320,-48.440,112.210,-0.0200,-0.0200,1.0000
C00553=56.410,-43.040,108.130,-0.0200,-0.0200,1.0000
C00554=51.460,-40.290,105.020,0.0200,0.1600,0.9900
C00555=47.690,-41.700,103.750,-0.2000,0.2700,0.9400
C00556=45.810,-43.560,103.700,-0.2600,0.2400,0.9400
C00557=44.690,-44.690,103.730,-0.2500,0.2500,0.9400
C00558=43.560,-45.810,103.700,-0.2400,0.2600,0.9400
C00559=41.700,-47.700,103.750,-0.2700,0.2000,0.9400
C00560=40.290,-51.460,105.020,-0.1600,-0.0200,0.9900
C00561=43.040,-56.410,108.130,0.0200,0.0200,1.0000
C00562=48.440,-63.320,112.210,0.0200,0.0200,1.0000
C00563=55.080,-71.840,116.120,0.0100,0.0100,1.0000
C00564=61.890,-80.660,118.910,0.0100,0.0000,1.0000
C00565=13.270,-100.800,118.910,-0.0100,-0.0000,1.0000
C00566=11.850,-89.740,116.120,-0.0200,-0.0000,1.0000
C00567=10.520,-79.020,112.210,-0.0300,-0.0000,1.0000
C00568=9.450,-70.320,108.130,-0.0300,-0.0000,1.0000
C00569=7.900,-64.870,105.020,0.1200,0.1000,0.9900
C00570=4.240,-63.210,103.750,0.0500,0.3300,0.9400
C00571=1.590,-63.200,103.700,-0.0100,0.3500,0.9400
C00572=0.000,-63.210,103.730,-0.0000,0.3500,0.9400
C00573=0.000,-63.210,103.730,-0.0000,0.3500,0.9400
C00574=-1.590,-63.200,103.700,0.0100,0.3500,0.9400
C00575=-4.240,-63.210,103.750,-0.0500,0.3300,0.9400
C00576=-7.900,-64.870,105.020,-0.1200,0.1000,0.9900
C00577=-9.450,-70.320,108.130,0.0300,-0.0000,1.0000
C00578=-10.520,-79.020,112.210,0.0300,-0.0000,1.0000
C00579=-11.850,-89.740,116.120,0.0200,-0.0000,1.0000
C00580=-13.270,-100.800,118.910,0.0100,-0.0000,1.0000
C00581=-61.890,-80.660,118.910,-0.0100,0.0000,1.0000
C00582=-55.080,-71.840,116.120,-0.0100,0.0100,1.0000
C00583=-48.440,-63.320,112.210,-0.0200,0.0200,1.0000
C00584=-43.040,-56.410,108.130,-0.0200,0.0200,1.0000
C00585=-40.290,-51.460,105.020,0.1600,-0.0200,0.9900
C00586=-41.700,-47.690,103.750,0.2700,0.2000,0.9400
C00587=-43.560,-45.810,103.700,0.2400,0.2600,0.9400
C00588=-44.690,-44.690,103.730,0.2500,0.2500,0.9400
C00589=-45.810,-43.560,103.700,0.2600,0.2400,0.9400
C00590=-47.700,-41.700,103.750,0.2000,0.2700,0.9400
C00591=-51.460,-40.290,105.020,-0.0200,0.1600,0.9900
C00592=-56.410,-43.040,108.130,0.0200,-0.0200,1.0000
C00593=-63.320,-48.440,112.210,0.0200,-0.0200,1.0000
C00594=-71.840,-55.080,116.120,0.0100,-0.0100,1.0000
C00595=-80.660,-61.890,118.910,0.0000,-0.0100,1.0000
C00596=-100.800,-13.270,118.910,-0.0000,0.0100,1.0000
C00597=-89.740,-11.850,116.120,-0.0000,0.0200,1.0000
C00598=-79.020,-10.520,112.210,-0.0000,0.0300,1.0000
C00599=-70.320,-9.450,108.130,-0.0000,0.0300,1.0000
C00600=-64.870,-7.900,105.020,0.1000,-0.1200,0.9900
C00601=-63.210,-4.240,103.750,0.3300,-0.0500,0.9400
C00602=-63.200,-1.590,103.700,0.3500,0.0100,0.9400
C00603=-63.210,0.000,103.730,0.3500,0.0000,0.9400
C00604=-63.200,1.590,103.700,0.3500,-0.0100,0.9400
C00605=-63.210,4.240,103.750,0.3300,0.0500,0.9400
C00606=-64.870,7.900,105.020,0.1000,0.1200,0.9900
C00607=-70.320,9.450,108.130,-0.0000,-0.0300,1.0000
C00608=-79.020,10.520,112.210,-0.0000,-0.0300,1.0000
C00609=-89.740,11.850,116.120,-0.0000,-0.0200,1.0000
C00610=-100.800,13.270,118.910,-0.0000,-0.0100,1.0000
C00611=-80.660,61.890,118.910,0.0000,0.0100,1.0000
C00612=-71.840,55.080,116.120,0.0100,0.0100,1.0000
C00613=-63.320,48.440,112.210,0.0200,0.0200,1.0000
C00614=-56.410,43.040,108.130,0.0200,0.0200,1.0000
C00615=-51.460,40.290,105.020,-0.0200,-0.1600,0.9900
C00616=-47.690,41.700,103.750,0.2000,-0.2700,0.9400
C00617=-45.810,43.560,103.700,0.2600,-0.2400,0.9400
C00618=-44.690,44.690,103.730,0.2500,-0.2500,0.9400
C00619=-43.560,45.810,103.700,0.2400,-0.2600,0.9400
C00620=-41.700,47.700,103.750,0.2700,-0.2000,0.9400
C00621=-40.290,51.460,105.020,0.1600,0.0200,0.9900
C00622=-43.040,56.410,108.130,-0.0200,-0.0200,1.0000
C00623=-48.440,63.320,112.210,-0.0200,-0.0200,1.0000
C00624=-55.080,71.840,116.120,-0.0100,-0.0100,1.0000
C00625=-61.890,80.660,118.910,-0.0100,-0.0000,1.0000
C00626=-13.270,100.800,118.910,0.0100,0.0000,1.0000
C00627=-11.850,89.740,116.120,0.0200,0.0000,1.0000
C00628=-10.520,79.020,112.210,0.0300,0.0000,1.0000
C00629=-9.450,70.320,108.130,0.0300,0.0000,1.0000
C00630=-7.900,64.870,105.020,-0.1200,-0.1000,0.9900
C00631=-4.240,63.210,103.750,-0.0500,-0.3300,0.9400
C00632=-1.590,63.200,103.700,0.0100,-0.3500,0.9400
C00633=0.000,63.210,103.730,-0.0000,-0.3500,0.9400
C00634=0.000,62.630,105.330,-0.0000,-0.3300,0.9500
C00635=-1.540,62.620,105.300,0.0100,-0.3300,0.9500
C00636=-4.150,62.640,105.350,-0.0500,-0.3100,0.9500
C00637=-7.800,64.360,106.640,-0.1100,-0.0900,0.9900
C00638=-9.350,69.950,109.790,0.0300,0.0000,1.0000
C00639=-10.450,78.820,113.900,0.0200,0.0000,1.0000
C00640=-11.820,89.670,117.820,0.0100,0.0000,1.0000
C00641=-55.050,71.770,117.820,-0.0100,-0.0100,1.0000
C00642=-48.350,63.130,113.900,-0.0200,-0.0100,1.0000
C00643=-42.850,56.080,109.790,-0.0200,-0.0200,1.0000
C00644=-40.000,51.030,106.640,0.1400,0.0100,0.9900
C00645=-41.360,47.230,105.350,0.2500,-0.1800,0.9500
C00646=-43.190,45.370,105.300,0.2200,-0.2400,0.9500
C00647=-44.290,44.290,105.330,0.2300,-0.2300,0.9500
C00648=-45.370,43.190,105.300,0.2400,-0.2200,0.9500
C00649=-47.230,41.360,105.350,0.1800,-0.2500,0.9500
C00650=-51.030,40.000,106.640,-0.0100,-0.1400,0.9900
C00651=-56.080,42.850,109.790,0.0200,0.0200,1.0000
C00652=-63.130,48.350,113.900,0.0100,0.0200,1.0000
C00653=-71.770,55.050,117.820,0.0100,0.0100,1.0000
C00654=-89.670,11.820,117.820,-0.0000,-0.0100,1.0000
C00655=-78.820,10.450,113.900,-0.0000,-0.0200,1.0000
C00656=-69.950,9.350,109.790,-0.0000,-0.0300,1.0000
C00657=-64.360,7.800,106.640,0.0900,0.1100,0.9900
C00658=-62.640,4.150,105.350,0.3100,0.0500,0.9500
C00659=-62.620,1.540,105.300,0.3300,-0.0100,0.9500
C00660=-62.630,0.000,105.330,0.3300,0.0000,0.9500
C00661=-62.620,-1.540,105.300,0.3300,0.0100,0.9500
C00662=-62.640,-4.150,105.350,0.3100,-0.0500,0.9500
C00663=-64.360,-7.800,106.640,0.0900,-0.1100,0.9900
C00664=-69.950,-9.350,109.790,-0.0000,0.0300,1.0000
C00665=-78.820,-10.450,113.900,-0.0000,0.0200,1.0000
C00666=-89.670,-11.820,117.820,-0.0000,0.0100,1.0000
C00667=-71.770,-55.050,117.820,0.0100,-0.0100,1.0000
C00668=-63.130,-48.350,113.900,0.0100,-0.0200,1.0000
C00669=-56.080,-42.850,109.790,0.0200,-0.0200,1.0000
C00670=-51.030,-40.000,106.640,-0.0100,0.1400,0.9900
C00671=-47.230,-41.360,105.350,0.1800,0.2500,0.9500
C00672=-45.370,-43.190,105.300,0.2400,0.2200,0.9500
C00673=-44.290,-44.290,105.330,0.2300,0.2300,0.9500
C00674=-43.190,-45.370,105.300,0.2200,0.2400,0.9500
C00675=-41.360,-47.230,105.350,0.2500,0.1800,0.9500
C00676=-40.000,-51.030,106.640,0.1400,-0.0100,0.9900
C00677=-42.850,-56.080,109.790,-0.0200,0.0200,1.0000
C00678=-48.350,-63.130,113.900,-0.0200,0.0100,1.0000
C00679=-55.050,-71.770,117.820,-0.0100,0.0100,1.0000
C00680=-11.820,-89.670,117.820,0.0100,-0.0000,1.0000
C00681=-10.450,-78.820,113.900,0.0200,-0.0000,1.0000
C00682=-9.350,-69.950,109.790,0.0300,-0.0000,1.0000
C00683=-7.800,-64.360,106.640,-0.1100,0.0900,0.9900
C00684=-4.150,-62.640,105.350,-0.0500,0.3100,0.9500
C00685=-1.540,-62.620,105.300,0.0100,0.3300,0.9500
C00686=0.000,-62.630,105.330,-0.0000,0.3300,0.9500
C00687=0.000,-62.630,105.330,-0.0000,0.3300,0.9500
C00688=1.540,-62.620,105.300,-0.0100,0.3300,0.9500
C00689=4.150,-62.640,105.350,0.0500,0.3100,0.9500
C00690=7.800,-64.360,106.640,0.1100,0.0900,0.9900
C00691=9.350,-69.950,109.790,-0.0300,-0.0000,1.0000
C00692=10.450,-78.820,113.900,-0.0200,-0.0000,1.0000
C00693=11.820,-89.670,117.820,-0.0100,-0.0000,1.0000
C00694=55.050,-71.770,117.820,0.0100,0.0100,1.0000
C00695=48.350,-63.130,113.900,0.0200,0.0100,1.0000
C00696=42.850,-56.080,109.790,0.0200,0.0200,1.0000
C00697=40.000,-51.030,106.640,-0.1400,-0.0100,0.9900
C00698=41.360,-47.230,105.350,-0.2500,0.1800,0.9500
C00699=43.190,-45.370,105.300,-0.2200,0.2400,0.9500
C00700=44.290,-44.290,105.330,-0.2300,0.2300,0.9500
C00701=45.370,-43.190,105.300,-0.2400,0.2200,0.9500
C00702=47.230,-41.360,105.350,-0.1800,0.2500,0.9500
C00703=51.030,-40.000,106.640,0.0100,0.1400,0.9900
C00704=56.080,-42.850,109.790,-0.0200,-0.0200,1.0000
C00705=63.130,-48.350,113.900,-0.0100,-0.0200,1.0000
C00706=71.770,-55.050,117.820,-0.0100,-0.0100,1.0000
C00707=89.670,-11.820,117.820,0.0000,0.0100,1.0000
C00708=78.820,-10.450,113.900,0.0000,0.0200,1.0000
C00709=69.950,-9.350,109.790,0.0000,0.0300,1.0000
C00710=64.360,-7.800,106.640,-0.0900,-0.1100,0.9900
C00711=62.640,-4.150,105.350,-0.3100,-0.0500,0.9500
C00712=62.620,-1.540,105.300,-0.3300,0.0100,0.9500
C00713=62.630,0.000,105.330,-0.3300,-0.0000,0.9500
C00714=62.620,1.540,105.300,-0.3300,-0.0100,0.9500
C00715=62.640,4.150,105.350,-0.3100,0.0500,0.9500
C00716=64.360,7.800,106.640,-0.0900,0.1100,0.9900
C00717=69.950,9.350,109.790,0.0000,-0.0300,1.0000
C00718=78.820,10.450,113.900,0.0000,-0.0200,1.0000
C00719=89.670,11.820,117.820,0.0000,-0.0100,1.0000
C00720=71.770,55.050,117.820,-0.0100,0.0100,1.0000
C00721=63.130,48.350,113.900,-0.0100,0.0200,1.0000
C00722=56.080,42.850,109.790,-0.0200,0.0200,1.0000
C00723=51.030,40.000,106.640,0.0100,-0.1400,0.9900
C00724=47.230,41.360,105.350,-0.1800,-0.2500,0.9500
C00725=45.370,43.190,105.300,-0.2400,-0.2200,0.9500
C00726=44.290,44.290,105.330,-0.2300,-0.2300,0.9500
C00727=43.190,45.370,105.300,-0.2200,-0.2400,0.9500
C00728=41.360,47.230,105.350,-0.2500,-0.1800,0.9500
C00729=40.000,51.030,106.640,-0.1400,0.0100,0.9900
C00730=42.850,56.080,109.790,0.0200,-0.0200,1.0000
C00731=48.350,63.130,113.900,0.0200,-0.0100,1.0000
C00732=55.050,71.770,117.820,0.0100,-0.0100,1.0000
C00733=11.820,89.670,117.820,-0.0100,0.0000,1.0000
C00734=10.450,78.820,113.900,-0.0200,0.0000,1.0000
C00735=9.350,69.950,109.790,-0.0300,0.0000,1.0000
C00736=7.800,64.360,106.640,0.1100,-0.0900,0.9900
C00737=4.150,62.640,105.350,0.0500,-0.3100,0.9500
C00738=1.540,62.620,105.300,-0.0100,-0.3300,0.9500
C00739=0.000,62.630,105.330,-0.0000,-0.3300,0.9500
C00740=0.000,62.100,106.950,-0.0000,-0.3000,0.9500
C00741=1.490,62.090,106.910,-0.0100,-0.3000,0.9500
C00742=4.070,62.120,106.970,0.0500,-0.2800,0.9600
C00743=7.710,63.900,108.270,0.1000,-0.0800,0.9900
C00744=9.270,69.630,111.460,-0.0200,0.0000,1.0000
C00745=10.400,78.670,115.590,-0.0200,0.0000,1.0000
C00746=11.800,89.640,119.520,-0.0000,0.0000,1.0000
C00747=55.040,71.730,119.520,0.0000,-0.0000,1.0000
C00748=48.280,62.980,115.590,0.0100,-0.0100,1.0000
C00749=42.680,55.790,111.460,0.0200,-0.0100,1.0000
C00750=39.740,50.630,108.270,-0.1200,0.0100,0.9900
C00751=41.050,46.800,106.970,-0.2300,-0.1600,0.9600
C00752=42.850,44.960,106.910,-0.2000,-0.2200,0.9500
C00753=43.910,43.910,106.950,-0.2100,-0.2100,0.9500
C00754=44.960,42.850,106.910,-0.2200,-0.2000,0.9500
C00755=46.800,41.050,106.970,-0.1600,-0.2300,0.9600
C00756=50.630,39.740,108.270,0.0100,-0.1200,0.9900
C00757=55.790,42.680,111.460,-0.0100,0.0200,1.0000
C00758=62.980,48.280,115.590,-0.0100,0.0100,1.0000
C00759=71.730,55.040,119.520,-0.0000,0.0000,1.0000
C00760=89.640,11.800,119.520,0.0000,-0.0000,1.0000
C00761=78.670,10.400,115.590,0.0000,-0.0200,1.0000
C00762=69.630,9.270,111.460,0.0000,-0.0200,1.0000
C00763=63.900,7.710,108.270,-0.0800,0.1000,0.9900
C00764=62.120,4.070,106.970,-0.2800,0.0500,0.9600
C00765=62.090,1.490,106.910,-0.3000,-0.0100,0.9500
C00766=62.100,0.000,106.950,-0.3000,-0.0000,0.9500
C00767=62.090,-1.490,106.910,-0.3000,0.0100,0.9500
C00768=62.120,-4.070,106.970,-0.2800,-0.0500,0.9600
C00769=63.900,-7.710,108.270,-0.0800,-0.1000,0.9900
C00770=69.630,-9.270,111.460,0.0000,0.0200,1.0000
C00771=78.670,-10.400,115.590,0.0000,0.0200,1.0000
C00772=89.640,-11.800,119.520,0.0000,0.0000,1.0000
C00773=71.730,-55.040,119.520,-0.0000,-0.0000,1.0000
C00774=62.980,-48.280,115.590,-0.0100,-0.0100,1.0000
C00775=55.790,-42.680,111.460,-0.0100,-0.0200,1.0000
C00776=50.630,-39.740,108.270,0.0100,0.1200,0.9900
C00777=46.800,-41.050,106.970,-0.1600,0.2300,0.9600
C00778=44.960,-42.850,106.910,-0.2200,0.2000,0.9500
C00779=43.910,-43.910,106.950,-0.2100,0.2100,0.9500
C00780=42.850,-44.960,106.910,-0.2000,0.2200,0.9500
C00781=41.050,-46.800,106.970,-0.2300,0.1600,0.9600
C00782=39.740,-50.630,108.270,-0.1200,-0.0100,0.9900
C00783=42.680,-55.790,111.460,0.0200,0.0100,1.0000
C00784=48.280,-62.980,115.590,0.0100,0.0100,1.0000
C00785=55.040,-71.730,119.520,0.0000,0.0000,1.0000
C00786=11.800,-89.640,119.520,-0.0000,-0.0000,1.0000
C00787=10.400,-78.670,115.590,-0.0200,-0.0000,1.0000
C00788=9.270,-69.630,111.460,-0.0200,-0.0000,1.0000
C00789=7.710,-63.900,108.270,0.1000,0.0800,0.9900
C00790=4.070,-62.120,106.970,0.0500,0.2800,0.9600
C00791=1.490,-62.090,106.910,-0.0100,0.3000,0.9500
C00792=0.000,-62.100,106.950,-0.0000,0.3000,0.9500
C00793=0.000,-62.100,106.950,-0.0000,0.3000,0.9500
C00794=-1.490,-62.090,106.910,0.0100,0.3000,0.9500
C00795=-4.070,-62.120,106.970,-0.0500,0.2800,0.9600
C00796=-7.710,-63.900,108.270,-0.1000,0.0800,0.9900
C00797=-9.270,-69.630,111.460,0.0200,-0.0000,1.0000
C00798=-10.400,-78.670,115.590,0.0200,-0.0000,1.0000
C00799=-11.800,-89.640,119.520,0.0000,-0.0000,1.0000
C00800=-55.040,-71.730,119.520,-0.0000,0.0000,1.0000
C00801=-48.280,-62.980,115.590,-0.0100,0.0100,1.0000
C00802=-42.680,-55.790,111.460,-0.0200,0.0100,1.0000
C00803=-39.740,-50.630,108.270,0.1200,-0.0100,0.9900
C00804=-41.050,-46.800,106.970,0.2300,0.1600,0.9600
C00805=-42.850,-44.960,106.910,0.2000,0.2200,0.9500
C00806=-43.910,-43.910,106.950,0.2100,0.2100,0.9500
C00807=-44.960,-42.850,106.910,0.2200,0.2000,0.9500
C00808=-46.800,-41.050,106.970,0.1600,0.2300,0.9600
C00809=-50.630,-39.740,108.270,-0.0100,0.1200,0.9900
C00810=-55.790,-42.680,111.460,0.0100,-0.0200,1.0000
C00811=-62.980,-48.280,115.590,0.0100,-0.0100,1.0000
C00812=-71.730,-55.040,119.520,0.0000,-0.0000,1.0000
C00813=-89.640,-11.800,119.520,-0.0000,0.0000,1.0000
C00814=-78.670,-10.400,115.590,-0.0000,0.0200,1.0000
C00815=-69.630,-9.270,111.460,-0.0000,0.0200,1.0000
C00816=-63.900,-7.710,108.270,0.0800,-0.1000,0.9900
C00817=-62.120,-4.070,106.970,0.2800,-0.0500,0.9600
C00818=-62.090,-1.490,106.910,0.3000,0.0100,0.9500
C00819=-62.100,0.000,106.950,0.3000,0.0000,0.9500
C00820=-62.090,1.490,106.910,0.3000,-0.0100,0.9500
C00821=-62.120,4.070,106.970,0.2800,0.0500,0.9600
C00822=-63.900,7.710,108.270,0.0800,0.1000,0.9900
C00823=-69.630,9.270,111.460,-0.0000,-0.0200,1.0000
C00824=-78.670,10.400,115.590,-0.0000,-0.0200,1.0000
C00825=-89.640,11.800,119.520,-0.0000,-0.0000,1.0000
C00826=-71.730,55.040,119.520,0.0000,0.0000,1.0000
C00827=-62.980,48.280,115.590,0.0100,0.0100,1.0000
C00828=-55.790,42.680,111.460,0.0100,0.0200,1.0000
C00829=-50.630,39.740,108.270,-0.0100,-0.1200,0.9900
C00830=-46.800,41.050,106.970,0.1600,-0.2300,0.9600
C00831=-44.960,42.850,106.910,0.2200,-0.2000,0.9500
C00832=-43.910,43.910,106.950,0.2100,-0.2100,0.9500
C00833=-42.850,44.960,106.910,0.2000,-0.2200,0.9500
C00834=-41.050,46.800,106.970,0.2300,-0.1600,0.9600
C00835=-39.740,50.630,108.270,0.1200,0.0100,0.9900
C00836=-42.680,55.790,111.460,-0.0200,-0.0100,1.0000
C00837=-48.280,62.980,115.590,-0.0100,-0.0100,1.0000
C00838=-55.040,71.730,119.520,-0.0000,-0.0000,1.0000
C00839=-11.800,89.640,119.520,0.0000,0.0000,1.0000
C00840=-10.400,78.670,115.590,0.0200,0.0000,1.0000
C00841=-9.270,69.630,111.460,0.0200,0.0000,1.0000
C00842=-7.710,63.900,108.270,-0.1000,-0.0800,0.9900
C00843=-4.070,62.120,106.970,-0.0500,-0.2800,0.9600
C00844=-1.490,62.090,106.910,0.0100,-0.3000,0.9500
C00845=0.000,62.100,106.950,-0.0000,-0.3000,0.9500
C00846=0.000,61.620,108.580,-0.0000,-0.2700,0.9600
C00847=-1.450,61.610,108.540,0.0100,-0.2700,0.9600
C00848=-4.000,61.650,108.600,-0.0400,-0.2500,0.9700
C00849=-7.630,63.490,109.920,-0.0800,-0.0700,0.9900
C00850=-9.200,69.360,113.130,0.0200,0.0000,1.0000
C00851=-10.360,78.560,117.290,0.0100,0.0000,1.0000
C00852=-48.230,62.880,117.290,-0.0100,-0.0100,1.0000
C00853=-42.540,55.550,113.130,-0.0100,-0.0100,1.0000
C00854=-39.500,50.290,109.920,0.1100,0.0100,0.9900
C00855=-40.770,46.420,108.600,0.2100,-0.1400,0.9700
C00856=-42.540,44.590,108.540,0.1800,-0.1900,0.9600
C00857=-43.570,43.570,108.580,0.1900,-0.1900,0.9600
C00858=-44.590,42.540,108.540,0.1900,-0.1800,0.9600
C00859=-46.420,40.770,108.600,0.1400,-0.2100,0.9700
C00860=-50.290,39.500,109.920,-0.0100,-0.1100,0.9900
C00861=-55.550,42.540,113.130,0.0100,0.0100,1.0000
C00862=-62.880,48.230,117.290,0.0100,0.0100,1.0000
C00863=-78.560,10.360,117.290,-0.0000,-0.0100,1.0000
C00864=-69.360,9.200,113.130,-0.0000,-0.0200,1.0000
C00865=-63.490,7.630,109.920,0.0700,0.0800,0.9900
C00866=-61.650,4.000,108.600,0.2500,0.0400,0.9700
C00867=-61.610,1.450,108.540,0.2700,-0.0100,0.9600
C00868=-61.620,0.000,108.580,0.2700,0.0000,0.9600
C00869=-61.610,-1.450,108.540,0.2700,0.0100,0.9600
C00870=-61.650,-4.000,108.600,0.2500,-0.0400,0.9700
C00871=-63.490,-7.630,109.920,0.0700,-0.0800,0.9900
C00872=-69.360,-9.200,113.130,-0.0000,0.0200,1.0000
C00873=-78.560,-10.360,117.290,-0.0000,0.0100,1.0000
C00874=-62.880,-48.230,117.290,0.0100,-0.0100,1.0000
C00875=-55.550,-42.540,113.130,0.0100,-0.0100,1.0000
C00876=-50.290,-39.500,109.920,-0.0100,0.1100,0.9900
C00877=-46.420,-40.770,108.600,0.1400,0.2100,0.9700
C00878=-44.590,-42.540,108.540,0.1900,0.1800,0.9600
C00879=-43.570,-43.570,108.580,0.1900,0.1900,0.9600
C00880=-42.540,-44.590,108.540,0.1800,0.1900,0.9600
C00881=-40.770,-46.420,108.600,0.2100,0.1400,0.9700
C00882=-39.500,-50.290,109.920,0.1100,-0.0100,0.9900
C00883=-42.540,-55.550,113.130,-0.0100,0.0100,1.0000
C00884=-48.230,-62.880,117.290,-0.0100,0.0100,1.0000
C00885=-10.360,-78.560,117.290,0.0100,-0.0000,1.0000
C00886=-9.200,-69.360,113.130,0.0200,-0.0000,1.0000
C00887=-7.630,-63.490,109.920,-0.0800,0.0700,0.9900
C00888=-4.000,-61.650,108.600,-0.0400,0.2500,0.9700
C00889=-1.450,-61.610,108.540,0.0100,0.2700,0.9600
C00890=0.000,-61.620,108.580,-0.0000,0.2700,0.9600
C00891=0.000,-61.620,108.580,-0.0000,0.2700,0.9600
C00892=1.450,-61.610,108.540,-0.0100,0.2700,0.9600
C00893=4.000,-61.650,108.600,0.0400,0.2500,0.9700
C00894=7.630,-63.490,109.920,0.0800,0.0700,0.9900
C00895=9.200,-69.360,113.130,-0.0200,-0.0000,1.0000
C00896=10.360,-78.560,117.290,-0.0100,-0.0000,1.0000
C00897=48.230,-62.880,117.290,0.0100,0.0100,1.0000
C00898=42.540,-55.550,113.130,0.0100,0.0100,1.0000
C00899=39.500,-50.290,109.920,-0.1100,-0.0100,0.9900
C00900=40.770,-46.420,108.600,-0.2100,0.1400,0.9700
C00901=42.540,-44.590,108.540,-0.1800,0.1900,0.9600
C00902=43.570,-43.570,108.580,-0.1900,0.1900,0.9600
C00903=44.590,-42.540,108.540,-0.1900,0.1800,0.9600
C00904=46.420,-40.770,108.600,-0.1400,0.2100,0.9700
C00905=50.290,-39.500,109.920,0.0100,0.1100,0.9900
C00906=55.550,-42.540,113.130,-0.0100,-0.0100,1.0000
C00907=62.880,-48.230,117.290,-0.0100,-0.0100,1.0000
C00908=78.560,-10.360,117.290,0.0000,0.0100,1.0000
C00909=69.360,-9.200,113.130,0.0000,0.0200,1.0000
C00910=63.490,-7.630,109.920,-0.0700,-0.0800,0.9900
C00911=61.650,-4.000,108.600,-0.2500,-0.0400,0.9700
C00912=61.610,-1.450,108.540,-0.2700,0.0100,0.9600
C00913=61.620,0.000,108.580,-0.2700,-0.0000,0.9600
C00914=61.610,1.450,108.540,-0.2700,-0.0100,0.9600
C00915=61.650,4.000,108.600,-0.2500,0.0400,0.9700
C00916=63.490,7.630,109.920,-0.0700,0.0800,0.9900
C00917=69.360,9.200,113.130,0.0000,-0.0200,1.0000
C00918=78.560,10.360,117.290,0.0000,-0.0100,1.0000
C00919=62.880,48.230,117.290,-0.0100,0.0100,1.0000
C00920=55.550,42.540,113.130,-0.0100,0.0100,1.0000
C00921=50.290,39.500,109.920,0.0100,-0.1100,0.9900
C00922=46.420,40.770,108.600,-0.1400,-0.2100,0.9700
C00923=44.590,42.540,108.540,-0.1900,-0.1800,0.9600
C00924=43.570,43.570,108.580,-0.1900,-0.1900,0.9600
C00925=42.540,44.590,108.540,-0.1800,-0.1900,0.9600
C00926=40.770,46.420,108.600,-0.2100,-0.1400,0.9700
C00927=39.500,50.290,109.920,-0.1100,0.0100,0.9900
C00928=42.540,55.550,113.130,0.0100,-0.0100,1.0000
C00929=48.230,62.880,117.290,0.0100,-0.0100,1.0000
C00930=10.360,78.560,117.290,-0.0100,0.0000,1.0000
C00931=9.200,69.360,113.130,-0.0200,0.0000,1.0000
C00932=7.630,63.490,109.920,0.0800,-0.0700,0.9900
C00933=4.000,61.650,108.600,0.0400,-0.2500,0.9700
C00934=1.450,61.610,108.540,-0.0100,-0.2700,0.9600
C00935=0.000,61.620,108.580,-0.0000,-0.2700,0.9600
C00936=0.000,61.200,110.230,-0.0000,-0.2300,0.9700
C00937=1.410,61.190,110.190,-0.0100,-0.2300,0.9700
C00938=3.930,61.230,110.250,0.0400,-0.2200,0.9800
C00939=7.550,63.140,111.580,0.0700,-0.0600,1.0000
C00940=9.140,69.150,114.820,-0.0100,0.0000,1.0000
C00941=10.340,78.510,118.990,-0.0000,0.0000,1.0000
C00942=48.200,62.820,118.990,0.0000,-0.0000,1.0000
C00943=42.430,55.360,114.820,0.0100,-0.0100,1.0000
C00944=39.300,49.990,111.580,-0.0900,0.0100,1.0000
C00945=40.520,46.080,110.250,-0.1800,-0.1300,0.9800
C00946=42.270,44.260,110.190,-0.1600,-0.1700,0.9700
C00947=43.270,43.270,110.230,-0.1600,-0.1600,0.9700
C00948=44.260,42.270,110.190,-0.1700,-0.1600,0.9700
C00949=46.080,40.520,110.250,-0.1300,-0.1800,0.9800
C00950=49.990,39.300,111.580,0.0100,-0.0900,1.0000
C00951=55.360,42.430,114.820,-0.0100,0.0100,1.0000
C00952=62.820,48.200,118.990,-0.0000,0.0000,1.0000
C00953=78.510,10.340,118.990,0.0000,-0.0000,1.0000
C00954=69.150,9.140,114.820,0.0000,-0.0100,1.0000
C00955=63.140,7.550,111.580,-0.0600,0.0700,1.0000
C00956=61.230,3.930,110.250,-0.2200,0.0400,0.9800
C00957=61.190,1.410,110.190,-0.2300,-0.0100,0.9700
C00958=61.200,0.000,110.230,-0.2300,-0.0000,0.9700
C00959=61.190,-1.410,110.190,-0.2300,0.0100,0.9700
C00960=61.230,-3.930,110.250,-0.2200,-0.0400,0.9800
C00961=63.140,-7.560,111.580,-0.0600,-0.0700,1.0000
C00962=69.150,-9.140,114.820,0.0000,0.0100,1.0000
C00963=78.510,-10.340,118.990,0.0000,0.0000,1.0000
C00964=62.820,-48.200,118.990,-0.0000,-0.0000,1.0000
C00965=55.360,-42.430,114.820,-0.0100,-0.0100,1.0000
C00966=49.990,-39.300,111.580,0.0100,0.0900,1.0000
C00967=46.080,-40.520,110.250,-0.1300,0.1800,0.9800
C00968=44.260,-42.270,110.190,-0.1700,0.1600,0.9700
C00969=43.270,-43.270,110.230,-0.1600,0.1600,0.9700
C00970=42.270,-44.260,110.190,-0.1600,0.1700,0.9700
C00971=40.520,-46.080,110.250,-0.1800,0.1300,0.9800
C00972=39.300,-49.990,111.580,-0.0900,-0.0100,1.0000
C00973=42.430,-55.360,114.820,0.0100,0.0100,1.0000
C00974=48.200,-62.820,118.990,0.0000,0.0000,1.0000
C00975=10.340,-78.510,118.990,-0.0000,-0.0000,1.0000
C00976=9.140,-69.150,114.820,-0.0100,-0.0000,1.0000
C00977=7.550,-63.140,111.580,0.0700,0.0600,1.0000
C00978=3.930,-61.230,110.250,0.0400,0.2200,0.9800
C00979=1.410,-61.190,110.190,-0.0100,0.2300,0.9700
C00980=0.000,-61.200,110.230,-0.0000,0.2300,0.9700
C00981=0.000,-61.200,110.230,-0.0000,0.2300,0.9700
C00982=-1.410,-61.190,110.190,0.0100,0.2300,0.9700
C00983=-3.930,-61.230,110.250,-0.0400,0.2200,0.9800
C00984=-7.560,-63.140,111.580,-0.0700,0.0600,1.0000
C00985=-9.140,-69.150,114.820,0.0100,-0.0000,1.0000
C00986=-10.340,-78.510,118.990,0.0000,-0.0000,1.0000
C00987=-48.200,-62.820,118.990,-0.0000,0.0000,1.0000
C00988=-42.430,-55.360,114.820,-0.0100,0.0100,1.0000
C00989=-39.300,-49.990,111.580,0.0900,-0.0100,1.0000
C00990=-40.520,-46.080,110.250,0.1800,0.1300,0.9800
C00991=-42.270,-44.260,110.190,0.1600,0.1700,0.9700
C00992=-43.270,-43.270,110.230,0.1600,0.1600,0.9700
C00993=-44.260,-42.270,110.190,0.1700,0.1600,0.9700
C00994=-46.080,-40.520,110.250,0.1300,0.1800,0.9800
C00995=-49.990,-39.300,111.580,-0.0100,0.0900,1.0000
C00996=-55.360,-42.430,114.820,0.0100,-0.0100,1.0000
C00997=-62.820,-48.200,118.990,0.0000,-0.0000,1.0000
C00998=-78.510,-10.340,118.990,-0.0000,0.0000,1.0000
C00999=-69.150,-9.140,114.820,-0.0000,0.0100,1.0000
C01000=-63.140,-7.550,111.580,0.0600,-0.0700,1.0000
C01001=-61.230,-3.930,110.250,0.2200,-0.0400,0.9800
C01002=-61.190,-1.410,110.190,0.2300,0.0100,0.9700
C01003=-61.200,0.000,110.230,0.2300,0.0000,0.9700
C01004=-61.190,1.410,110.190,0.2300,-0.0100,0.9700
C01005=-61.230,3.930,110.250,0.2200,0.0400,0.9800
C01006=-63.140,7.560,111.580,0.0600,0.0700,1.0000
C01007=-69.150,9.140,114.820,-0.0000,-0.0100,1.0000
C01008=-78.510,10.340,118.990,-0.0000,-0.0000,1.0000
C01009=-62.820,48.200,118.990,0.0000,0.0000,1.0000
C01010=-55.360,42.430,114.820,0.0100,0.0100,1.0000
C01011=-49.990,39.300,111.580,-0.0100,-0.0900,1.0000
C01012=-46.080,40.520,110.250,0.1300,-0.1800,0.9800
C01013=-44.260,42.270,110.190,0.1700,-0.1600,0.9700
C01014=-43.270,43.270,110.230,0.1600,-0.1600,0.9700
C01015=-42.270,44.260,110.190,0.1600,-0.1700,0.9700
C01016=-40.520,46.080,110.250,0.1800,-0.1300,0.9800
C01017=-39.300,49.990,111.580,0.0900,0.0100,1.0000
C01018=-42.430,55.360,114.820,-0.0100,-0.0100,1.0000
C01019=-48.200,62.820,118.990,-0.0000,-0.0000,1.0000
C01020=-10.340,78.510,118.990,0.0000,0.0000,1.0000
C01021=-9.140,69.150,114.820,0.0100,0.0000,1.0000
C01022=-7.560,63.140,111.580,-0.0700,-0.0600,1.0000
C01023=-3.930,61.230,110.250,-0.0400,-0.2200,0.9800
C01024=-1.410,61.190,110.190,0.0100,-0.2300,0.9700
C01025=0.000,61.200,110.230,-0.0000,-0.2300,0.9700
C01026=0.000,60.830,111.890,-0.0000,-0.2000,0.9800
C01027=-1.380,60.820,111.850,0.0000,-0.2000,0.9800
C01028=-3.880,60.870,111.910,-0.0300,-0.1800,0.9800
C01029=-7.500,62.840,113.250,-0.0600,-0.0400,1.0000
C01030=-9.100,68.990,116.510,0.0100,0.0000,1.0000
C01031=-42.350,55.220,116.510,-0.0100,-0.0100,1.0000
C01032=-39.130,49.730,113.250,0.0700,0.0100,1.0000
C01033=-40.300,45.780,111.910,0.1500,-0.1100,0.9800
C01034=-42.040,43.980,111.850,0.1400,-0.1400,0.9800
C01035=-43.020,43.020,111.890,0.1400,-0.1400,0.9800
C01036=-43.980,42.040,111.850,0.1400,-0.1400,0.9800
C01037=-45.780,40.300,111.910,0.1100,-0.1500,0.9800
C01038=-49.730,39.130,113.250,-0.0100,-0.0700,1.0000
C01039=-55.220,42.350,116.510,0.0100,0.0100,1.0000
C01040=-68.990,9.100,116.510,-0.0000,-0.0100,1.0000
C01041=-62.840,7.500,113.250,0.0400,0.0600,1.0000
C01042=-60.870,3.880,111.910,0.1800,0.0300,0.9800
C01043=-60.820,1.380,111.850,0.2000,-0.0000,0.9800
C01044=-60.830,0.000,111.890,0.2000,0.0000,0.9800
C01045=-60.820,-1.380,111.850,0.2000,0.0000,0.9800
C01046=-60.870,-3.870,111.910,0.1800,-0.0300,0.9800
C01047=-62.840,-7.500,113.250,0.0400,-0.0600,1.0000
C01048=-68.990,-9.100,116.510,-0.0000,0.0100,1.0000
C01049=-55.220,-42.350,116.510,0.0100,-0.0100,1.0000
C01050=-49.730,-39.130,113.250,-0.0100,0.0700,1.0000
C01051=-45.780,-40.300,111.910,0.1100,0.1500,0.9800
C01052=-43.980,-42.040,111.850,0.1400,0.1400,0.9800
C01053=-43.020,-43.020,111.890,0.1400,0.1400,0.9800
C01054=-42.040,-43.980,111.850,0.1400,0.1400,0.9800
C01055=-40.300,-45.780,111.910,0.1500,0.1100,0.9800
C01056=-39.130,-49.730,113.250,0.0700,-0.0100,1.0000
C01057=-42.350,-55.220,116.510,-0.0100,0.0100,1.0000
C01058=-9.100,-68.990,116.510,0.0100,-0.0000,1.0000
C01059=-7.500,-62.840,113.250,-0.0600,0.0400,1.0000
C01060=-3.880,-60.870,111.910,-0.0300,0.1800,0.9800
C01061=-1.380,-60.820,111.850,0.0000,0.2000,0.9800
C01062=0.000,-60.830,111.890,-0.0000,0.2000,0.9800
C01063=0.000,-60.830,111.890,-0.0000,0.2000,0.9800
C01064=1.380,-60.820,111.850,-0.0000,0.2000,0.9800
C01065=3.870,-60.870,111.910,0.0300,0.1800,0.9800
C01066=7.500,-62.840,113.250,0.0600,0.0400,1.0000
C01067=9.100,-68.990,116.510,-0.0100,-0.0000,1.0000
C01068=42.350,-55.220,116.510,0.0100,0.0100,1.0000
C01069=39.130,-49.730,113.250,-0.0700,-0.0100,1.0000
C01070=40.300,-45.780,111.910,-0.1500,0.1100,0.9800
C01071=42.040,-43.980,111.850,-0.1400,0.1400,0.9800
C01072=43.020,-43.020,111.890,-0.1400,0.1400,0.9800
C01073=43.980,-42.040,111.850,-0.1400,0.1400,0.9800
C01074=45.780,-40.300,111.910,-0.1100,0.1500,0.9800
C01075=49.730,-39.130,113.250,0.0100,0.0700,1.0000
C01076=55.220,-42.350,116.510,-0.0100,-0.0100,1.0000
C01077=68.990,-9.100,116.510,0.0000,0.0100,1.0000
C01078=62.840,-7.500,113.250,-0.0400,-0.0600,1.0000
C01079=60.870,-3.880,111.910,-0.1800,-0.0300,0.9800
C01080=60.820,-1.380,111.850,-0.2000,0.0000,0.9800
C01081=60.830,0.000,111.890,-0.2000,-0.0000,0.9800
C01082=60.820,1.380,111.850,-0.2000,-0.0000,0.9800
C01083=60.870,3.870,111.910,-0.1800,0.0300,0.9800
C01084=62.840,7.500,113.250,-0.0400,0.0600,1.0000
C01085=68.990,9.100,116.510,0.0000,-0.0100,1.0000
C01086=55.220,42.350,116.510,-0.0100,0.0100,1.0000
C01087=49.730,39.130,113.250,0.0100,-0.0700,1.0000
C01088=45.780,40.300,111.910,-0.1100,-0.1500,0.9800
C01089=43.980,42.040,111.850,-0.1400,-0.1400,0.9800
C01090=43.020,43.020,111.890,-0.1400,-0.1400,0.9800
C01091=42.040,43.980,111.850,-0.1400,-0.1400,0.9800
C01092=40.300,45.780,111.910,-0.1500,-0.1100,0.9800
C01093=39.130,49.730,113.250,-0.0700,0.0100,1.0000
C01094=42.350,55.220,116.510,0.0100,-0.0100,1.0000
C01095=9.100,68.990,116.510,-0.0100,0.0000,1.0000
C01096=7.500,62.840,113.250,0.0600,-0.0400,1.0000
C01097=3.870,60.870,111.910,0.0300,-0.1800,0.9800
C01098=1.380,60.820,111.850,-0.0000,-0.2000,0.9800
C01099=0.000,60.830,111.890,-0.0000,-0.2000,0.9800
C01100=0.000,60.530,113.560,-0.0000,-0.1600,0.9900
C01101=1.350,60.520,113.520,-0.0000,-0.1600,0.9900
C01102=3.830,60.570,113.580,0.0300,-0.1500,0.9900
C01103=7.450,62.600,114.940,0.0400,-0.0300,1.0000
C01104=9.070,68.900,118.210,-0.0100,0.0000,1.0000
C01105=42.300,55.130,118.210,0.0000,-0.0000,1.0000
C01106=39.000,49.530,114.940,-0.0500,0.0100,1.0000
C01107=40.120,45.540,113.580,-0.1200,-0.0900,0.9900
C01108=41.840,43.750,113.520,-0.1100,-0.1200,0.9900
C01109=42.800,42.800,113.560,-0.1100,-0.1100,0.9900
C01110=43.750,41.840,113.520,-0.1200,-0.1100,0.9900
C01111=45.540,40.120,113.580,-0.0900,-0.1200,0.9900
C01112=49.530,39.000,114.940,0.0100,-0.0500,1.0000
C01113=55.130,42.300,118.210,-0.0000,0.0000,1.0000
C01114=68.900,9.070,118.210,0.0000,-0.0100,1.0000
C01115=62.600,7.450,114.940,-0.0300,0.0400,1.0000
C01116=60.570,3.830,113.580,-0.1500,0.0300,0.9900
C01117=60.520,1.350,113.520,-0.1600,-0.0000,0.9900
C01118=60.530,0.000,113.560,-0.1600,-0.0000,0.9900
C01119=60.520,-1.350,113.520,-0.1600,0.0000,0.9900
C01120=60.570,-3.830,113.580,-0.1500,-0.0300,0.9900
C01121=62.600,-7.450,114.940,-0.0300,-0.0400,1.0000
C01122=68.900,-9.070,118.210,0.0000,0.0100,1.0000
C01123=55.130,-42.300,118.210,-0.0000,-0.0000,1.0000
C01124=49.530,-39.000,114.940,0.0100,0.0500,1.0000
C01125=45.540,-40.120,113.580,-0.0900,0.1200,0.9900
C01126=43.750,-41.840,113.520,-0.1200,0.1100,0.9900
C01127=42.800,-42.800,113.560,-0.1100,0.1100,0.9900
C01128=41.840,-43.750,113.520,-0.1100,0.1200,0.9900
C01129=40.120,-45.540,113.580,-0.1200,0.0900,0.9900
C01130=39.000,-49.530,114.940,-0.0500,-0.0100,1.0000
C01131=42.300,-55.130,118.210,0.0000,0.0000,1.0000
C01132=9.070,-68.900,118.210,-0.0100,-0.0000,1.0000
C01133=7.450,-62.600,114.940,0.0400,0.0300,1.0000
C01134=3.830,-60.570,113.580,0.0300,0.1500,0.9900
C01135=1.350,-60.520,113.520,-0.0000,0.1600,0.9900
C01136=0.000,-60.530,113.560,-0.0000,0.1600,0.9900
C01137=0.000,-60.530,113.560,-0.0000,0.1600,0.9900
C01138=-1.350,-60.520,113.520,0.0000,0.1600,0.9900
C01139=-3.830,-60.570,113.580,-0.0300,0.1500,0.9900
C01140=-7.450,-62.600,114.940,-0.0400,0.0300,1.0000
C01141=-9.070,-68.900,118.210,0.0100,-0.0000,1.0000
C01142=-42.300,-55.130,118.210,-0.0000,0.0000,1.0000
C01143=-39.000,-49.530,114.940,0.0500,-0.0100,1.0000
C01144=-40.120,-45.540,113.580,0.1200,0.0900,0.9900
C01145=-41.840,-43.750,113.520,0.1100,0.1200,0.9900
C01146=-42.800,-42.800,113.560,0.1100,0.1100,0.9900
C01147=-43.750,-41.840,113.520,0.1200,0.1100,0.9900
C01148=-45.540,-40.120,113.580,0.0900,0.1200,0.9900
C01149=-49.530,-39.000,114.940,-0.0100,0.0500,1.0000
C01150=-55.130,-42.300,118.210,0.0000,-0.0000,1.0000
C01151=-68.900,-9.070,118.210,-0.0000,0.0100,1.0000
C01152=-62.600,-7.450,114.940,0.0300,-0.0400,1.0000
C01153=-60.570,-3.830,113.580,0.1500,-0.0300,0.9900
C01154=-60.520,-1.350,113.520,0.1600,0.0000,0.9900
C01155=-60.530,0.000,113.560,0.1600,0.0000,0.9900
C01156=-60.520,1.350,113.520,0.1600,-0.0000,0.9900
C01157=-60.570,3.830,113.580,0.1500,0.0300,0.9900
C01158=-62.600,7.450,114.940,0.0300,0.0400,1.0000
C01159=-68.900,9.070,118.210,-0.0000,-0.0100,1.0000
C01160=-55.130,42.300,118.210,0.0000,0.0000,1.0000
C01161=-49.530,39.000,114.940,-0.0100,-0.0500,1.0000
C01162=-45.540,40.120,113.580,0.0900,-0.1200,0.9900
C01163=-43.750,41.840,113.520,0.1200,-0.1100,0.9900
C01164=-42.800,42.800,113.560,0.1100,-0.1100,0.9900
C01165=-41.840,43.750,113.520,0.1100,-0.1200,0.9900
C01166=-40.120,45.540,113.580,0.1200,-0.0900,0.9900
C01167=-39.000,49.530,114.940,0.0500,0.0100,1.0000
C01168=-42.300,55.130,118.210,-0.0000,-0.0000,1.0000
C01169=-9.070,68.900,118.210,0.0100,0.0000,1.0000
C01170=-7.450,62.600,114.940,-0.0400,-0.0300,1.0000
C01171=-3.830,60.570,113.580,-0.0300,-0.1500,0.9900
C01172=-1.350,60.520,113.520,0.0000,-0.1600,0.9900
C01173=0.000,60.530,113.560,-0.0000,-0.1600,0.9900
C01174=0.000,60.290,115.240,-0.0000,-0.1200,0.9900
C01175=-1.330,60.280,115.200,0.0000,-0.1200,0.9900
C01176=-3.790,60.340,115.260,-0.0200,-0.1100,0.9900
C01177=-7.420,62.430,116.630,-0.0300,-0.0200,1.0000
C01178=-9.070,68.860,119.910,0.0000,0.0000,1.0000
C01179=-42.280,55.100,119.910,-0.0000,-0.0000,1.0000
C01180=-38.900,49.390,116.630,0.0400,0.0000,1.0000
C01181=-39.980,45.350,115.260,0.0900,-0.0600,0.9900
C01182=-41.690,43.560,115.200,0.0800,-0.0900,0.9900
C01183=-42.630,42.630,115.240,0.0800,-0.0800,0.9900
C01184=-43.560,41.690,115.200,0.0900,-0.0800,0.9900
C01185=-45.350,39.980,115.260,0.0600,-0.0900,0.9900
C01186=-49.390,38.900,116.630,-0.0000,-0.0400,1.0000
C01187=-55.100,42.280,119.910,0.0000,0.0000,1.0000
C01188=-68.860,9.070,119.910,-0.0000,-0.0000,1.0000
C01189=-62.430,7.420,116.630,0.0200,0.0300,1.0000
C01190=-60.340,3.790,115.260,0.1100,0.0200,0.9900
C01191=-60.280,1.330,115.200,0.1200,-0.0000,0.9900
C01192=-60.290,0.000,115.240,0.1200,0.0000,0.9900
C01193=-60.280,-1.330,115.200,0.1200,0.0000,0.9900
C01194=-60.340,-3.790,115.260,0.1100,-0.0200,0.9900
C01195=-62.430,-7.420,116.630,0.0200,-0.0300,1.0000
C01196=-68.860,-9.070,119.910,-0.0000,0.0000,1.0000
C01197=-55.100,-42.280,119.910,0.0000,-0.0000,1.0000
C01198=-49.390,-38.900,116.630,-0.0000,0.0400,1.0000
C01199=-45.350,-39.980,115.260,0.0600,0.0900,0.9900
C01200=-43.560,-41.690,115.200,0.0900,0.0800,0.9900
C01201=-42.630,-42.630,115.240,0.0800,0.0800,0.9900
C01202=-41.690,-43.560,115.200,0.0800,0.0900,0.9900
C01203=-39.980,-45.350,115.260,0.0900,0.0600,0.9900
C01204=-38.900,-49.390,116.630,0.0400,-0.0000,1.0000
C01205=-42.280,-55.100,119.910,-0.0000,0.0000,1.0000
C01206=-9.070,-68.860,119.910,0.0000,-0.0000,1.0000
C01207=-7.420,-62.430,116.630,-0.0300,0.0200,1.0000
C01208=-3.790,-60.340,115.260,-0.0200,0.1100,0.9900
C01209=-1.330,-60.280,115.200,0.0000,0.1200,0.9900
C01210=0.000,-60.290,115.240,-0.0000,0.1200,0.9900
C01211=0.000,-60.290,115.240,-0.0000,0.1200,0.9900
C01212=1.330,-60.280,115.200,-0.0000,0.1200,0.9900
C01213=3.790,-60.340,115.260,0.0200,0.1100,0.9900
C01214=7.420,-62.430,116.630,0.0300,0.0200,1.0000
C01215=9.070,-68.860,119.910,-0.0000,-0.0000,1.0000
C01216=42.280,-55.100,119.910,0.0000,0.0000,1.0000
C01217=38.900,-49.390,116.630,-0.0400,-0.0000,1.0000
C01218=39.980,-45.350,115.260,-0.0900,0.0600,0.9900
C01219=41.690,-43.560,115.200,-0.0800,0.0900,0.9900
C01220=42.630,-42.630,115.240,-0.0800,0.0800,0.9900
C01221=43.560,-41.690,115.200,-0.0900,0.0800,0.9900
C01222=45.350,-39.980,115.260,-0.0600,0.0900,0.9900
C01223=49.390,-38.900,116.630,0.0000,0.0400,1.0000
C01224=55.100,-42.280,119.910,-0.0000,-0.0000,1.0000
C01225=68.860,-9.070,119.910,0.0000,0.0000,1.0000
C01226=62.430,-7.420,116.630,-0.0200,-0.0300,1.0000
C01227=60.340,-3.790,115.260,-0.1100,-0.0200,0.9900
C01228=60.280,-1.330,115.200,-0.1200,0.0000,0.9900
C01229=60.290,0.000,115.240,-0.1200,-0.0000,0.9900
C01230=60.280,1.330,115.200,-0.1200,-0.0000,0.9900
C01231=60.340,3.790,115.260,-0.1100,0.0200,0.9900
C01232=62.430,7.420,116.630,-0.0200,0.0300,1.0000
C01233=68.860,9.070,119.910,0.0000,-0.0000,1.0000
C01234=55.100,42.280,119.910,-0.0000,0.0000,1.0000
C01235=49.390,38.900,116.630,0.0000,-0.0400,1.0000
C01236=45.350,39.980,115.260,-0.0600,-0.0900,0.9900
C01237=43.560,41.690,115.200,-0.0900,-0.0800,0.9900
C01238=42.630,42.630,115.240,-0.0800,-0.0800,0.9900
C01239=41.690,43.560,115.200,-0.0800,-0.0900,0.9900
C01240=39.980,45.350,115.260,-0.0900,-0.0600,0.9900
C01241=38.900,49.390,116.630,-0.0400,0.0000,1.0000
C01242=42.280,55.100,119.910,0.0000,-0.0000,1.0000
C01243=9.070,68.860,119.910,-0.0000,0.0000,1.0000
C01244=7.420,62.430,116.630,0.0300,-0.0200,1.0000
C01245=3.790,60.340,115.260,0.0200,-0.1100,0.9900
C01246=1.330,60.280,115.200,-0.0000,-0.1200,0.9900
C01247=0.000,60.290,115.240,-0.0000,-0.1200,0.9900
C01248=0.000,60.120,116.930,-0.0000,-0.0800,1.0000
C01249=1.310,60.110,116.890,-0.0000,-0.0800,1.0000
C01250=3.770,60.170,116.950,0.0100,-0.0700,1.0000
C01251=7.400,62.330,118.320,0.0100,-0.0100,1.0000
C01252=38.840,49.300,118.320,-0.0200,0.0000,1.0000
C01253=39.880,45.210,116.950,-0.0600,-0.0400,1.0000
C01254=41.580,43.430,116.890,-0.0600,-0.0600,1.0000
C01255=42.510,42.510,116.930,-0.0600,-0.0600,1.0000
C01256=43.430,41.580,116.890,-0.0600,-0.0600,1.0000
C01257=45.210,39.880,116.950,-0.0400,-0.0600,1.0000
C01258=49.300,38.840,118.320,0.0000,-0.0200,1.0000
C01259=62.330,7.400,118.320,-0.0100,0.0100,1.0000
C01260=60.170,3.770,116.950,-0.0700,0.0100,1.0000
C01261=60.110,1.310,116.890,-0.0800,-0.0000,1.0000
C01262=60.120,0.000,116.930,-0.0800,-0.0000,1.0000
C01263=60.110,-1.310,116.890,-0.0800,0.0000,1.0000
C01264=60.170,-3.770,116.950,-0.0700,-0.0100,1.0000
C01265=62.330,-7.400,118.320,-0.0100,-0.0100,1.0000
C01266=49.300,-38.840,118.320,0.0000,0.0200,1.0000
C01267=45.210,-39.880,116.950,-0.0400,0.0600,1.0000
C01268=43.430,-41.580,116.890,-0.0600,0.0600,1.0000
C01269=42.510,-42.510,116.930,-0.0600,0.0600,1.0000
C01270=41.580,-43.430,116.890,-0.0600,0.0600,1.0000
C01271=39.880,-45.210,116.950,-0.0600,0.0400,1.0000
C01272=38.840,-49.300,118.320,-0.0200,-0.0000,1.0000
C01273=7.400,-62.330,118.320,0.0100,0.0100,1.0000
C01274=3.770,-60.170,116.950,0.0100,0.0700,1.0000
C01275=1.310,-60.110,116.890,-0.0000,0.0800,1.0000
C01276=0.000,-60.120,116.930,-0.0000,0.0800,1.0000
C01277=0.000,-60.120,116.930,-0.0000,0.0800,1.0000
C01278=-1.310,-60.110,116.890,0.0000,0.0800,1.0000
C01279=-3.770,-60.170,116.950,-0.0100,0.0700,1.0000
C01280=-7.400,-62.330,118.320,-0.0100,0.0100,1.0000
C01281=-38.840,-49.300,118.320,0.0200,-0.0000,1.0000
C01282=-39.880,-45.210,116.950,0.0600,0.0400,1.0000
C01283=-41.580,-43.430,116.890,0.0600,0.0600,1.0000
C01284=-42.510,-42.510,116.930,0.0600,0.0600,1.0000
C01285=-43.430,-41.580,116.890,0.0600,0.0600,1.0000
C01286=-45.210,-39.880,116.950,0.0400,0.0600,1.0000
C01287=-49.300,-38.840,118.320,-0.0000,0.0200,1.0000
C01288=-62.330,-7.400,118.320,0.0100,-0.0100,1.0000
C01289=-60.170,-3.770,116.950,0.0700,-0.0100,1.0000
C01290=-60.110,-1.310,116.890,0.0800,0.0000,1.0000
C01291=-60.120,0.000,116.930,0.0800,0.0000,1.0000
C01292=-60.110,1.310,116.890,0.0800,-0.0000,1.0000
C01293=-60.170,3.770,116.950,0.0700,0.0100,1.0000
C01294=-62.330,7.400,118.320,0.0100,0.0100,1.0000
C01295=-49.300,38.840,118.320,-0.0000,-0.0200,1.0000
C01296=-45.210,39.880,116.950,0.0400,-0.0600,1.0000
C01297=-43.430,41.580,116.890,0.0600,-0.0600,1.0000
C01298=-42.510,42.510,116.930,0.0600,-0.0600,1.0000
C01299=-41.580,43.430,116.890,0.0600,-0.0600,1.0000
C01300=-39.880,45.210,116.950,0.0600,-0.0400,1.0000
C01301=-38.840,49.300,118.320,0.0200,0.0000,1.0000
C01302=-7.400,62.330,118.320,-0.0100,-0.0100,1.0000
C01303=-3.770,60.170,116.950,-0.0100,-0.0700,1.0000
C01304=-1.310,60.110,116.890,0.0000,-0.0800,1.0000
C01305=0.000,60.120,116.930,-0.0000,-0.0800,1.0000
C01306=0.000,60.020,118.630,-0.0000,-0.0400,1.0000
C01307=-1.300,60.010,118.590,0.0000,-0.0400,1.0000
C01308=-3.750,60.080,118.650,-0.0100,-0.0300,1.0000
C01309=-39.830,45.130,118.650,0.0300,-0.0200,1.0000
C01310=-41.520,43.350,118.590,0.0300,-0.0300,1.0000
C01311=-42.440,42.440,118.630,0.0300,-0.0300,1.0000
C01312=-43.360,41.510,118.590,0.0300,-0.0300,1.0000
C01313=-45.130,39.830,118.650,0.0200,-0.0300,1.0000
C01314=-60.080,3.750,118.650,0.0300,0.0100,1.0000
C01315=-60.010,1.300,118.590,0.0400,-0.0000,1.0000
C01316=-60.020,0.000,118.630,0.0400,0.0000,1.0000
C01317=-60.010,-1.300,118.590,0.0400,0.0000,1.0000
C01318=-60.080,-3.750,118.650,0.0300,-0.0100,1.0000
C01319=-45.130,-39.830,118.650,0.0200,0.0300,1.0000
C01320=-43.350,-41.520,118.590,0.0300,0.0300,1.0000
C01321=-42.440,-42.440,118.630,0.0300,0.0300,1.0000
C01322=-41.510,-43.360,118.590,0.0300,0.0300,1.0000
C01323=-39.830,-45.130,118.650,0.0300,0.0200,1.0000
C01324=-3.750,-60.080,118.650,-0.0100,0.0300,1.0000
C01325=-1.300,-60.010,118.590,0.0000,0.0400,1.0000
C01326=0.000,-60.020,118.630,-0.0000,0.0400,1.0000
C01327=0.000,-60.020,118.630,-0.0000,0.0400,1.0000
C01328=1.300,-60.010,118.590,-0.0000,0.0400,1.0000
C01329=3.750,-60.080,118.650,0.0100,0.0300,1.0000
C01330=39.830,-45.130,118.650,-0.0300,0.0200,1.0000
C01331=41.520,-43.350,118.590,-0.0300,0.0300,1.0000
C01332=42.440,-42.440,118.630,-0.0300,0.0300,1.0000
C01333=43.360,-41.510,118.590,-0.0300,0.0300,1.0000
C01334=45.130,-39.830,118.650,-0.0200,0.0300,1.0000
C01335=60.080,-3.750,118.650,-0.0300,-0.0100,1.0000
C01336=60.010,-1.300,118.590,-0.0400,0.0000,1.0000
C01337=60.020,0.000,118.630,-0.0400,-0.0000,1.0000
C01338=60.010,1.300,118.590,-0.0400,-0.0000,1.0000
C01339=60.080,3.750,118.650,-0.0300,0.0100,1.0000
C01340=45.130,39.830,118.650,-0.0200,-0.0300,1.0000
C01341=43.350,41.520,118.590,-0.0300,-0.0300,1.0000
C01342=42.440,42.440,118.630,-0.0300,-0.0300,1.0000
C01343=41.510,43.360,118.590,-0.0300,-0.0300,1.0000
C01344=39.830,45.130,118.650,-0.0300,-0.0200,1.0000
C01345=3.750,60.080,118.650,0.0100,-0.0300,1.0000
C01346=1.300,60.010,118.590,-0.0000,-0.0400,1.0000
C01347=0.000,60.020,118.630,-0.0000,-0.0400,1.0000
//INST
///DATE 03/29/2021 17:02
///COMM
///ATTR SC,RW,RJ
///FRAME ROBOT
///GROUP1 RB1
NOP
MOVL C00001
MOVL C00002
MOVL C00003
MOVL C00004
MOVL C00005
MOVL C00006
MOVL C00007
MOVL C00008
MOVL C00009
MOVL C00010
MOVL C00011
MOVL C00012
MOVL C00013
MOVL C00014
MOVL C00015
MOVL C00016
MOVL C00017
MOVL C00018
MOVL C00019
MOVL C00020
MOVL C00021
MOVL C00022
MOVL C00023
MOVL C00024
MOVL C00025
MOVL C00026
MOVL C00027
MOVL C00028
MOVL C00029
MOVL C00030
MOVL C00031
MOVL C00032
MOVL C00033
MOVL C00034
MOVL C00035
MOVL C00036
MOVL C00037
MOVL C00038
MOVL C00039
MOVL C00040
MOVL C00041
MOVL C00042
MOVL C00043
MOVL C00044
MOVL C00045
MOVL C00046
MOVL C00047
MOVL C00048
MOVL C00049
MOVL C00050
MOVL C00051
MOVL C00052
MOVL C00053
MOVL C00054
MOVL C00055
MOVL C00056
MOVL C00057
MOVL C00058
MOVL C00059
MOVL C00060
MOVL C00061
MOVL C00062
MOVL C00063
MOVL C00064
MOVL C00065
MOVL C00066
MOVL C00067
MOVL C00068
MOVL C00069
MOVL C00070
MOVL C00071
MOVL C00072
MOVL C00073
MOVL C00074
MOVL C00075
MOVL C00076
MOVL C00077
MOVL C00078
MOVL C00079
MOVL C00080
MOVL C00081
MOVL C00082
MOVL C00083
MOVL C00084
MOVL C00085
MOVL C00086
MOVL C00087
MOVL C00088
MOVL C00089
MOVL C00090
MOVL C00091
MOVL C00092
MOVL C00093
MOVL C00094
MOVL C00095
MOVL C00096
MOVL C00097
MOVL C00098
MOVL C00099
MOVL C00100
MOVL C00101
MOVL C00102
MOVL C00103
MOVL C00104
MOVL C00105
MOVL C00106
MOVL C00107
MOVL C00108
MOVL C00109
MOVL C00110
MOVL C00111
MOVL C00112
MOVL C00113
MOVL C00114
MOVL C00115
MOVL C00116
MOVL C00117
MOVL C00118
MOVL C00119
MOVL C00120
MOVL C00121
MOVL C00122
MOVL C00123
MOVL C00124
MOVL C00125
MOVL C00126
MOVL C00127
MOVL C00128
MOVL C00129
MOVL C00130
MOVL C00131
MOVL C00132
MOVL C00133
MOVL C00134
MOVL C00135
MOVL C00136
MOVL C00137
MOVL C00138
MOVL C00139
MOVL C00140
MOVL C00141
MOVL C00142
MOVL C00143
MOVL C00144
MOVL C00145
MOVL C00146
MOVL C00147
MOVL C00148
MOVL C00149
MOVL C00150
MOVL C00151
MOVL C00152
MOVL C00153
MOVL C00154
MOVL C00155
MOVL C00156
MOVL C00157
MOVL C00158
MOVL C00159
MOVL C00160
MOVL C00161
MOVL C00162
MOVL C00163
MOVL C00164
MOVL C00165
MOVL C00166
MOVL C00167
MOVL C00168
MOVL C00169
MOVL C00170
MOVL C00171
MOVL C00172
MOVL C00173
MOVL C00174
MOVL C00175
MOVL C00176
MOVL C00177
MOVL C00178
MOVL C00179
MOVL C00180
MOVL C00181
MOVL C00182
MOVL C00183
MOVL C00184
MOVL C00185
MOVL C00186
MOVL C00187
MOVL C00188
MOVL C00189
MOVL C00190
MOVL C00191
MOVL C00192
MOVL C00193
MOVL C00194
MOVL C00195
MOVL C00196
MOVL C00197
MOVL C00198
MOVL C00199
MOVL C00200
MOVL C00201
MOVL C00202
MOVL C00203
MOVL C00204
MOVL C00205
MOVL C00206
MOVL C00207
MOVL C00208
MOVL C00209
MOVL C00210
MOVL C00211
MOVL C00212
MOVL C00213
MOVL C00214
MOVL C00215
MOVL C00216
MOVL C00217
MOVL C00218
MOVL C00219
MOVL C00220
MOVL C00221
MOVL C00222
MOVL C00223
MOVL C00224
MOVL C00225
MOVL C00226
MOVL C00227
MOVL C00228
MOVL C00229
MOVL C00230
MOVL C00231
MOVL C00232
MOVL C00233
MOVL C00234
MOVL C00235
MOVL C00236
MOVL C00237
MOVL C00238
MOVL C00239
MOVL C00240
MOVL C00241
MOVL C00242
MOVL C00243
MOVL C00244
MOVL C00245
MOVL C00246
MOVL C00247
MOVL C00248
MOVL C00249
MOVL C00250
MOVL C00251
MOVL C00252
MOVL C00253
MOVL C00254
MOVL C00255
MOVL C00256
MOVL C00257
MOVL C00258
MOVL C00259
MOVL C00260
MOVL C00261
MOVL C00262
MOVL C00263
MOVL C00264
MOVL C00265
MOVL C00266
MOVL C00267
MOVL C00268
MOVL C00269
MOVL C00270
MOVL C00271
MOVL C00272
MOVL C00273
MOVL C00274
MOVL C00275
MOVL C00276
MOVL C00277
MOVL C00278
MOVL C00279
MOVL C00280
MOVL C00281
MOVL C00282
MOVL C00283
MOVL C00284
MOVL C00285
MOVL C00286
MOVL C00287
MOVL C00288
MOVL C00289
MOVL C00290
MOVL C00291
MOVL C00292
MOVL C00293
MOVL C00294
MOVL C00295
MOVL C00296
MOVL C00297
MOVL C00298
MOVL C00299
MOVL C00300
MOVL C00301
MOVL C00302
MOVL C00303
MOVL C00304
MOVL C00305
MOVL C00306
MOVL C00307
MOVL C00308
MOVL C00309
MOVL C00310
MOVL C00311
MOVL C00312
MOVL C00313
MOVL C00314
MOVL C00315
MOVL C00316
MOVL C00317
MOVL C00318
MOVL C00319
MOVL C00320
MOVL C00321
MOVL C00322
MOVL C00323
MOVL C00324
MOVL C00325
MOVL C00326
MOVL C00327
MOVL C00328
MOVL C00329
MOVL C00330
MOVL C00331
MOVL C00332
MOVL C00333
MOVL C00334
MOVL C00335
MOVL C00336
MOVL C00337
MOVL C00338
MOVL C00339
MOVL C00340
MOVL C00341
MOVL C00342
MOVL C00343
MOVL C00344
MOVL C00345
MOVL C00346
MOVL C00347
MOVL C00348
MOVL C00349
MOVL C00350
MOVL C00351
MOVL C00352
MOVL C00353
MOVL C00354
MOVL C00355
MOVL C00356
MOVL C00357
MOVL C00358
MOVL C00359
MOVL C00360
MOVL C00361
MOVL C00362
MOVL C00363
MOVL C00364
MOVL C00365
MOVL C00366
MOVL C00367
MOVL C00368
MOVL C00369
MOVL C00370
MOVL C00371
MOVL C00372
MOVL C00373
MOVL C00374
MOVL C00375
MOVL C00376
MOVL C00377
MOVL C00378
MOVL C00379
MOVL C00380
MOVL C00381
MOVL C00382
MOVL C00383
MOVL C00384
MOVL C00385
MOVL C00386
MOVL C00387
MOVL C00388
MOVL C00389
MOVL C00390
MOVL C00391
MOVL C00392
MOVL C00393
MOVL C00394
MOVL C00395
MOVL C00396
MOVL C00397
MOVL C00398
MOVL C00399
MOVL C00400
MOVL C00401
MOVL C00402
MOVL C00403
MOVL C00404
MOVL C00405
MOVL C00406
MOVL C00407
MOVL C00408
MOVL C00409
MOVL C00410
MOVL C00411
MOVL C00412
MOVL C00413
MOVL C00414
MOVL C00415
MOVL C00416
MOVL C00417
MOVL C00418
MOVL C00419
MOVL C00420
MOVL C00421
MOVL C00422
MOVL C00423
MOVL C00424
MOVL C00425
MOVL C00426
MOVL C00427
MOVL C00428
MOVL C00429
MOVL C00430
MOVL C00431
MOVL C00432
MOVL C00433
MOVL C00434
MOVL C00435
MOVL C00436
MOVL C00437
MOVL C00438
MOVL C00439
MOVL C00440
MOVL C00441
MOVL C00442
MOVL C00443
MOVL C00444
MOVL C00445
MOVL C00446
MOVL C00447
MOVL C00448
MOVL C00449
MOVL C00450
MOVL C00451
MOVL C00452
MOVL C00453
MOVL C00454
MOVL C00455
MOVL C00456
MOVL C00457
MOVL C00458
MOVL C00459
MOVL C00460
MOVL C00461
MOVL C00462
MOVL C00463
MOVL C00464
MOVL C00465
MOVL C00466
MOVL C00467
MOVL C00468
MOVL C00469
MOVL C00470
MOVL C00471
MOVL C00472
MOVL C00473
MOVL C00474
MOVL C00475
MOVL C00476
MOVL C00477
MOVL C00478
MOVL C00479
MOVL C00480
MOVL C00481
MOVL C00482
MOVL C00483
MOVL C00484
MOVL C00485
MOVL C00486
MOVL C00487
MOVL C00488
MOVL C00489
MOVL C00490
MOVL C00491
MOVL C00492
MOVL C00493
MOVL C00494
MOVL C00495
MOVL C00496
MOVL C00497
MOVL C00498
MOVL C00499
MOVL C00500
MOVL C00501
MOVL C00502
MOVL C00503
MOVL C00504
MOVL C00505
MOVL C00506
MOVL C00507
MOVL C00508
MOVL C00509
MOVL C00510
MOVL C00511
MOVL C00512
MOVL C00513
MOVL C00514
MOVL C00515
MOVL C00516
MOVL C00517
MOVL C00518
MOVL C00519
MOVL C00520
MOVL C00521
MOVL C00522
MOVL C00523
MOVL C00524
MOVL C00525
MOVL C00526
MOVL C00527
MOVL C00528
MOVL C00529
MOVL C00530
MOVL C00531
MOVL C00532
MOVL C00533
MOVL C00534
MOVL C00535
MOVL C00536
MOVL C00537
MOVL C00538
MOVL C00539
MOVL C00540
MOVL C00541
MOVL C00542
MOVL C00543
MOVL C00544
MOVL C00545
MOVL C00546
MOVL C00547
MOVL C00548
MOVL C00549
MOVL C00550
MOVL C00551
MOVL C00552
MOVL C00553
MOVL C00554
MOVL C00555
MOVL C00556
MOVL C00557
MOVL C00558
MOVL C00559
MOVL C00560
MOVL C00561
MOVL C00562
MOVL C00563
MOVL C00564
MOVL C00565
MOVL C00566
MOVL C00567
MOVL C00568
MOVL C00569
MOVL C00570
MOVL C00571
MOVL C00572
MOVL C00573
MOVL C00574
MOVL C00575
MOVL C00576
MOVL C00577
MOVL C00578
MOVL C00579
MOVL C00580
MOVL C00581
MOVL C00582
MOVL C00583
MOVL C00584
MOVL C00585
MOVL C00586
MOVL C00587
MOVL C00588
MOVL C00589
MOVL C00590
MOVL C00591
MOVL C00592
MOVL C00593
MOVL C00594
MOVL C00595
MOVL C00596
MOVL C00597
MOVL C00598
MOVL C00599
MOVL C00600
MOVL C00601
MOVL C00602
MOVL C00603
MOVL C00604
MOVL C00605
MOVL C00606
MOVL C00607
MOVL C00608
MOVL C00609
MOVL C00610
MOVL C00611
MOVL C00612
MOVL C00613
MOVL C00614
MOVL C00615
MOVL C00616
MOVL C00617
MOVL C00618
MOVL C00619
MOVL C00620
MOVL C00621
MOVL C00622
MOVL C00623
MOVL C00624
MOVL C00625
MOVL C00626
MOVL C00627
MOVL C00628
MOVL C00629
MOVL C00630
MOVL C00631
MOVL C00632
MOVL C00633
MOVL C00634
MOVL C00635
MOVL C00636
MOVL C00637
MOVL C00638
MOVL C00639
MOVL C00640
MOVL C00641
MOVL C00642
MOVL C00643
MOVL C00644
MOVL C00645
MOVL C00646
MOVL C00647
MOVL C00648
MOVL C00649
MOVL C00650
MOVL C00651
MOVL C00652
MOVL C00653
MOVL C00654
MOVL C00655
MOVL C00656
MOVL C00657
MOVL C00658
MOVL C00659
MOVL C00660
MOVL C00661
MOVL C00662
MOVL C00663
MOVL C00664
MOVL C00665
MOVL C00666
MOVL C00667
MOVL C00668
MOVL C00669
MOVL C00670
MOVL C00671
MOVL C00672
MOVL C00673
MOVL C00674
MOVL C00675
MOVL C00676
MOVL C00677
MOVL C00678
MOVL C00679
MOVL C00680
MOVL C00681
MOVL C00682
MOVL C00683
MOVL C00684
MOVL C00685
MOVL C00686
MOVL C00687
MOVL C00688
MOVL C00689
MOVL C00690
MOVL C00691
MOVL C00692
MOVL C00693
MOVL C00694
MOVL C00695
MOVL C00696
MOVL C00697
MOVL C00698
MOVL C00699
MOVL C00700
MOVL C00701
MOVL C00702
MOVL C00703
MOVL C00704
MOVL C00705
MOVL C00706
MOVL C00707
MOVL C00708
MOVL C00709
MOVL C00710
MOVL C00711
MOVL C00712
MOVL C00713
MOVL C00714
MOVL C00715
MOVL C00716
MOVL C00717
MOVL C00718
MOVL C00719
MOVL C00720
MOVL C00721
MOVL C00722
MOVL C00723
MOVL C00724
MOVL C00725
MOVL C00726
MOVL C00727
MOVL C00728
MOVL C00729
MOVL C00730
MOVL C00731
MOVL C00732
MOVL C00733
MOVL C00734
MOVL C00735
MOVL C00736
MOVL C00737
MOVL C00738
MOVL C00739
MOVL C00740
MOVL C00741
MOVL C00742
MOVL C00743
MOVL C00744
MOVL C00745
MOVL C00746
MOVL C00747
MOVL C00748
MOVL C00749
MOVL C00750
MOVL C00751
MOVL C00752
MOVL C00753
MOVL C00754
MOVL C00755
MOVL C00756
MOVL C00757
MOVL C00758
MOVL C00759
MOVL C00760
MOVL C00761
MOVL C00762
MOVL C00763
MOVL C00764
MOVL C00765
MOVL C00766
MOVL C00767
MOVL C00768
MOVL C00769
MOVL C00770
MOVL C00771
MOVL C00772
MOVL C00773
MOVL C00774
MOVL C00775
MOVL C00776
MOVL C00777
MOVL C00778
MOVL C00779
MOVL C00780
MOVL C00781
MOVL C00782
MOVL C00783
MOVL C00784
MOVL C00785
MOVL C00786
MOVL C00787
MOVL C00788
MOVL C00789
MOVL C00790
MOVL C00791
MOVL C00792
MOVL C00793
MOVL C00794
MOVL C00795
MOVL C00796
MOVL C00797
MOVL C00798
MOVL C00799
MOVL C00800
MOVL C00801
MOVL C00802
MOVL C00803
MOVL C00804
MOVL C00805
MOVL C00806
MOVL C00807
MOVL C00808
MOVL C00809
MOVL C00810
MOVL C00811
MOVL C00812
MOVL C00813
MOVL C00814
MOVL C00815
MOVL C00816
MOVL C00817
MOVL C00818
MOVL C00819
MOVL C00820
MOVL C00821
MOVL C00822
MOVL C00823
MOVL C00824
MOVL C00825
MOVL C00826
MOVL C00827
MOVL C00828
MOVL C00829
MOVL C00830
MOVL C00831
MOVL C00832
MOVL C00833
MOVL C00834
MOVL C00835
MOVL C00836
MOVL C00837
MOVL C00838
MOVL C00839
MOVL C00840
MOVL C00841
MOVL C00842
MOVL C00843
MOVL C00844
MOVL C00845
MOVL C00846
MOVL C00847
MOVL C00848
MOVL C00849
MOVL C00850
MOVL C00851
MOVL C00852
MOVL C00853
MOVL C00854
MOVL C00855
MOVL C00856
MOVL C00857
MOVL C00858
MOVL C00859
MOVL C00860
MOVL C00861
MOVL C00862
MOVL C00863
MOVL C00864
MOVL C00865
MOVL C00866
MOVL C00867
MOVL C00868
MOVL C00869
MOVL C00870
MOVL C00871
MOVL C00872
MOVL C00873
MOVL C00874
MOVL C00875
MOVL C00876
MOVL C00877
MOVL C00878
MOVL C00879
MOVL C00880
MOVL C00881
MOVL C00882
MOVL C00883
MOVL C00884
MOVL C00885
MOVL C00886
MOVL C00887
MOVL C00888
MOVL C00889
MOVL C00890
MOVL C00891
MOVL C00892
MOVL C00893
MOVL C00894
MOVL C00895
MOVL C00896
MOVL C00897
MOVL C00898
MOVL C00899
MOVL C00900
MOVL C00901
MOVL C00902
MOVL C00903
MOVL C00904
MOVL C00905
MOVL C00906
MOVL C00907
MOVL C00908
MOVL C00909
MOVL C00910
MOVL C00911
MOVL C00912
MOVL C00913
MOVL C00914
MOVL C00915
MOVL C00916
MOVL C00917
MOVL C00918
MOVL C00919
MOVL C00920
MOVL C00921
MOVL C00922
MOVL C00923
MOVL C00924
MOVL C00925
MOVL C00926
MOVL C00927
MOVL C00928
MOVL C00929
MOVL C00930
MOVL C00931
MOVL C00932
MOVL C00933
MOVL C00934
MOVL C00935
MOVL C00936
MOVL C00937
MOVL C00938
MOVL C00939
MOVL C00940
MOVL C00941
MOVL C00942
MOVL C00943
MOVL C00944
MOVL C00945
MOVL C00946
MOVL C00947
MOVL C00948
MOVL C00949
MOVL C00950
MOVL C00951
MOVL C00952
MOVL C00953
MOVL C00954
MOVL C00955
MOVL C00956
MOVL C00957
MOVL C00958
MOVL C00959
MOVL C00960
MOVL C00961
MOVL C00962
MOVL C00963
MOVL C00964
MOVL C00965
MOVL C00966
MOVL C00967
MOVL C00968
MOVL C00969
MOVL C00970
MOVL C00971
MOVL C00972
MOVL C00973
MOVL C00974
MOVL C00975
MOVL C00976
MOVL C00977
MOVL C00978
MOVL C00979
MOVL C00980
MOVL C00981
MOVL C00982
MOVL C00983
MOVL C00984
MOVL C00985
MOVL C00986
MOVL C00987
MOVL C00988
MOVL C00989
MOVL C00990
MOVL C00991
MOVL C00992
MOVL C00993
MOVL C00994
MOVL C00995
MOVL C00996
MOVL C00997
MOVL C00998
MOVL C00999
MOVL C01000
MOVL C01001
MOVL C01002
MOVL C01003
MOVL C01004
MOVL C01005
MOVL C01006
MOVL C01007
MOVL C01008
MOVL C01009
MOVL C01010
MOVL C01011
MOVL C01012
MOVL C01013
MOVL C01014
MOVL C01015
MOVL C01016
MOVL C01017
MOVL C01018
MOVL C01019
MOVL C01020
MOVL C01021
MOVL C01022
MOVL C01023
MOVL C01024
MOVL C01025
MOVL C01026
MOVL C01027
MOVL C01028
MOVL C01029
MOVL C01030
MOVL C01031
MOVL C01032
MOVL C01033
MOVL C01034
MOVL C01035
MOVL C01036
MOVL C01037
MOVL C01038
MOVL C01039
MOVL C01040
MOVL C01041
MOVL C01042
MOVL C01043
MOVL C01044
MOVL C01045
MOVL C01046
MOVL C01047
MOVL C01048
MOVL C01049
MOVL C01050
MOVL C01051
MOVL C01052
MOVL C01053
MOVL C01054
MOVL C01055
MOVL C01056
MOVL C01057
MOVL C01058
MOVL C01059
MOVL C01060
MOVL C01061
MOVL C01062
MOVL C01063
MOVL C01064
MOVL C01065
MOVL C01066
MOVL C01067
MOVL C01068
MOVL C01069
MOVL C01070
MOVL C01071
MOVL C01072
MOVL C01073
MOVL C01074
MOVL C01075
MOVL C01076
MOVL C01077
MOVL C01078
MOVL C01079
MOVL C01080
MOVL C01081
MOVL C01082
MOVL C01083
MOVL C01084
MOVL C01085
MOVL C01086
MOVL C01087
MOVL C01088
MOVL C01089
MOVL C01090
MOVL C01091
MOVL C01092
MOVL C01093
MOVL C01094
MOVL C01095
MOVL C01096
MOVL C01097
MOVL C01098
MOVL C01099
MOVL C01100
MOVL C01101
MOVL C01102
MOVL C01103
MOVL C01104
MOVL C01105
MOVL C01106
MOVL C01107
MOVL C01108
MOVL C01109
MOVL C01110
MOVL C01111
MOVL C01112
MOVL C01113
MOVL C01114
MOVL C01115
MOVL C01116
MOVL C01117
MOVL C01118
MOVL C01119
MOVL C01120
MOVL C01121
MOVL C01122
MOVL C01123
MOVL C01124
MOVL C01125
MOVL C01126
MOVL C01127
MOVL C01128
MOVL C01129
MOVL C01130
MOVL C01131
MOVL C01132
MOVL C01133
MOVL C01134
MOVL C01135
MOVL C01136
MOVL C01137
MOVL C01138
MOVL C01139
MOVL C01140
MOVL C01141
MOVL C01142
MOVL C01143
MOVL C01144
MOVL C01145
MOVL C01146
MOVL C01147
MOVL C01148
MOVL C01149
MOVL C01150
MOVL C01151
MOVL C01152
MOVL C01153
MOVL C01154
MOVL C01155
MOVL C01156
MOVL C01157
MOVL C01158
MOVL C01159
MOVL C01160
MOVL C01161
MOVL C01162
MOVL C01163
MOVL C01164
MOVL C01165
MOVL C01166
MOVL C01167
MOVL C01168
MOVL C01169
MOVL C01170
MOVL C01171
MOVL C01172
MOVL C01173
MOVL C01174
MOVL C01175
MOVL C01176
MOVL C01177
MOVL C01178
MOVL C01179
MOVL C01180
MOVL C01181
MOVL C01182
MOVL C01183
MOVL C01184
MOVL C01185
MOVL C01186
MOVL C01187
MOVL C01188
MOVL C01189
MOVL C01190
MOVL C01191
MOVL C01192
MOVL C01193
MOVL C01194
MOVL C01195
MOVL C01196
MOVL C01197
MOVL C01198
MOVL C01199
MOVL C01200
MOVL C01201
MOVL C01202
MOVL C01203
MOVL C01204
MOVL C01205
MOVL C01206
MOVL C01207
MOVL C01208
MOVL C01209
MOVL C01210
MOVL C01211
MOVL C01212
MOVL C01213
MOVL C01214
MOVL C01215
MOVL C01216
MOVL C01217
MOVL C01218
MOVL C01219
MOVL C01220
MOVL C01221
MOVL C01222
MOVL C01223
MOVL C01224
MOVL C01225
MOVL C01226
MOVL C01227
MOVL C01228
MOVL C01229
MOVL C01230
MOVL C01231
MOVL C01232
MOVL C01233
MOVL C01234
MOVL C01235
MOVL C01236
MOVL C01237
MOVL C01238
MOVL C01239
MOVL C01240
MOVL C01241
MOVL C01242
MOVL C01243
MOVL C01244
MOVL C01245
MOVL C01246
MOVL C01247
MOVL C01248
MOVL C01249
MOVL C01250
MOVL C01251
MOVL C01252
MOVL C01253
MOVL C01254
MOVL C01255
MOVL C01256
MOVL C01257
MOVL C01258
MOVL C01259
MOVL C01260
MOVL C01261
MOVL C01262
MOVL C01263
MOVL C01264
MOVL C01265
MOVL C01266
MOVL C01267
MOVL C01268
MOVL C01269
MOVL C01270
MOVL C01271
MOVL C01272
MOVL C01273
MOVL C01274
MOVL C01275
MOVL C01276
MOVL C01277
MOVL C01278
MOVL C01279
MOVL C01280
MOVL C01281
MOVL C01282
MOVL C01283
MOVL C01284
MOVL C01285
MOVL C01286
MOVL C01287
MOVL C01288
MOVL C01289
MOVL C01290
MOVL C01291
MOVL C01292
MOVL C01293
MOVL C01294
MOVL C01295
MOVL C01296
MOVL C01297
MOVL C01298
MOVL C01299
MOVL C01300
MOVL C01301
MOVL C01302
MOVL C01303
MOVL C01304
MOVL C01305
MOVL C01306
MOVL C01307
MOVL C01308
MOVL C01309
MOVL C01310
MOVL C01311
MOVL C01312
MOVL C01313
MOVL C01314
MOVL C01315
MOVL C01316
MOVL C01317
MOVL C01318
MOVL C01319
MOVL C01320
MOVL C01321
MOVL C01322
MOVL C01323
MOVL C01324
MOVL C01325
MOVL C01326
MOVL C01327
MOVL C01328
MOVL C01329
MOVL C01330
MOVL C01331
MOVL C01332
MOVL C01333
MOVL C01334
MOVL C01335
MOVL C01336
MOVL C01337
MOVL C01338
MOVL C01339
MOVL C01340
MOVL C01341
MOVL C01342
MOVL C01343
MOVL C01344
MOVL C01345
MOVL C01346
MOVL C01347
MOVL C01348
END
